KUKA KRL program: MyProgram_059().src

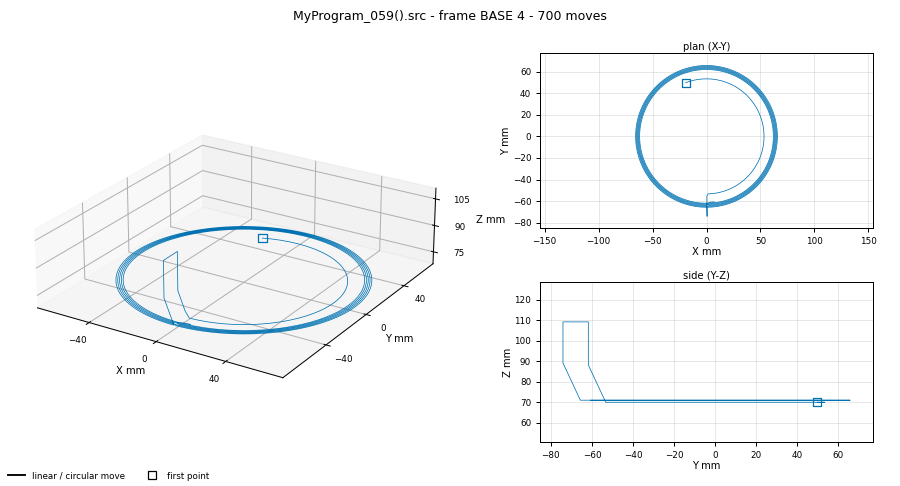
[picture p0: tool path of MyProgram_059().src in frame BASE 4, 700 of 700 moves have a stored position in this frame; points joined in program order, loops and branches not executed]
&ACCESS RVP
&REL 1
&PARAM TEMPLATE = C:\KRC\Roboter\Template\vorgabe
&PARAM EDITMASK = *
DEF MyProgram_059()
; ---- Setting reference (Base) ----
$BASE = BASE_DATA[4]

; --------------------------
; ---- Setting tool (TCP) ----
$TOOL = TOOL_DATA[3]
; --------------------------

$VEL.CP = VEL_APROX_PRINT
Startdeposition()
$VEL.CP = VEL_PRINT
LIN {X -19.2783,Y 49.7039,Z 70,A 103.8,B 24.8517,C -2.8098,E1 24.9442,E2 -20.1582} C_DIS
LIN {X -16.8217,Y 50.5882,Z 70,A 100.9889,B 24.8513,C -2.8131,E1 24.9516,E2 -17.3495} C_DIS
LIN {X -14.3168,Y 51.3533,Z 70,A 98.5431,B 24.8504,C -2.8223,E1 24.9581,E2 -14.9218} C_DIS
LIN {X -12.3251,Y 51.8679,Z 70,A 95.999,B 24.8507,C -2.8187,E1 24.9651,E2 -12.3655} C_DIS
LIN {X -9.9491,Y 52.3747,Z 70,A 93.3434,B 24.8506,C -2.8201,E1 24.9723,E2 -9.7102} C_DIS
LIN {X -7.1522,Y 52.8301,Z 70,A 90.3456,B 24.8503,C -2.8229,E1 24.9806,E2 -6.7165} C_DIS
LIN {X -4.5627,Y 53.1165,Z 70,A 87.5334,B 24.8502,C -2.8241,E1 24.9884,E2 -3.9056} C_DIS
LIN {X -2.028,Y 53.2732,Z 70,A 84.746,B 24.8502,C -2.8241,E1 24.9962,E2 -1.1173} C_DIS
LIN {X 0.6631,Y 53.308,Z 70,A 81.9222,B 24.85,C -2.8259,E1 25.0041,E2 1.7022} C_DIS
LIN {X 2.7693,Y 53.2395,Z 70,A 79.6668,B 24.85,C -2.8262,E1 25.0103,E2 3.9561} C_DIS
LIN {X 5.1925,Y 53.0585,Z 70,A 76.9708,B 24.8501,C -2.8244,E1 25.0178,E2 6.6547} C_DIS
LIN {X 7.8477,Y 52.7313,Z 70,A 74.1797,B 24.8501,C -2.8253,E1 25.0256,E2 9.4415} C_DIS
LIN {X 10.3045,Y 52.3063,Z 70,A 71.4304,B 24.8503,C -2.823,E1 25.0331,E2 12.1931} C_DIS
LIN {X 12.9755,Y 51.7089,Z 70,A 68.5235,B 24.8503,C -2.8221,E1 25.041,E2 15.0981} C_DIS
LIN {X 15.3915,Y 51.0415,Z 70,A 65.8321,B 24.8506,C -2.8203,E1 25.0482,E2 17.7892} C_DIS
LIN {X 17.8688,Y 50.2279,Z 70,A 63.0346,B 24.8508,C -2.818,E1 25.0556,E2 20.5865} C_DIS
LIN {X 20.3041,Y 49.2937,Z 70,A 60.2375,B 24.8511,C -2.8154,E1 25.0629,E2 23.3837} C_DIS
LIN {X 22.6903,Y 48.2418,Z 70,A 57.4092,B 24.8515,C -2.8117,E1 25.0701,E2 26.2135} C_DIS
LIN {X 25.039,Y 47.0657,Z 70,A 54.5794,B 24.8519,C -2.808,E1 25.0771,E2 29.0443} C_DIS
LIN {X 27.3333,Y 45.7715,Z 70,A 51.8043,B 24.8522,C -2.8051,E1 25.0838,E2 31.8179} C_DIS
LIN {X 29.6243,Y 44.3236,Z 70,A 48.9325,B 24.8526,C -2.8014,E1 25.0905,E2 34.6891} C_DIS
LIN {X 31.7582,Y 42.8206,Z 70,A 46.1065,B 24.8531,C -2.7963,E1 25.0969,E2 37.5173} C_DIS
LIN {X 33.7767,Y 41.2467,Z 70,A 43.3667,B 24.8536,C -2.7915,E1 25.1029,E2 40.2581} C_DIS
LIN {X 35.7658,Y 39.5343,Z 70,A 40.5427,B 24.8542,C -2.786,E1 25.1088,E2 43.0839} C_DIS
LIN {X 37.7091,Y 37.6855,Z 70,A 37.6907,B 24.8548,C -2.7807,E1 25.1145,E2 45.9366} C_DIS
LIN {X 39.4732,Y 35.8333,Z 70,A 34.9527,B 24.8554,C -2.775,E1 25.1197,E2 48.6762} C_DIS
LIN {X 41.1795,Y 33.8587,Z 70,A 32.1622,B 24.856,C -2.7689,E1 25.1248,E2 51.4684} C_DIS
LIN {X 42.8175,Y 31.7623,Z 70,A 29.318,B 24.8567,C -2.7624,E1 25.1296,E2 54.3145} C_DIS
LIN {X 44.3203,Y 29.6293,Z 70,A 26.559,B 24.8573,C -2.7563,E1 25.1339,E2 57.0741} C_DIS
LIN {X 45.6739,Y 27.496,Z 70,A 23.8275,B 24.8581,C -2.749,E1 25.138,E2 59.8092} C_DIS
LIN {X 46.9787,Y 25.202,Z 70,A 20.9748,B 24.8589,C -2.7411,E1 25.1418,E2 62.6655} C_DIS
LIN {X 48.1969,Y 22.7868,Z 70,A 18.1531,B 24.8595,C -2.7349,E1 25.1453,E2 65.4868} C_DIS
LIN {X 49.2137,Y 20.4974,Z 70,A 15.4462,B 24.8603,C -2.7271,E1 25.1483,E2 68.1975} C_DIS
LIN {X 50.191,Y 17.9733,Z 70,A 12.5854,B 24.8611,C -2.7197,E1 25.1511,E2 71.0598} C_DIS
LIN {X 50.9578,Y 15.6652,Z 70,A 10.2725,B 24.8612,C -2.7184,E1 25.153,E2 73.3627} C_DIS
LIN {X 51.5403,Y 13.6293,Z 70,A 7.7203,B 24.8625,C -2.7058,E1 25.1549,E2 75.9301} C_DIS
LIN {X 52.135,Y 11.1389,Z 70,A 4.9326,B 24.8634,C -2.6967,E1 25.1567,E2 78.7231} C_DIS
LIN {X 52.635,Y 8.4702,Z 70,A 2.0944,B 24.8642,C -2.6894,E1 25.158,E2 81.5619} C_DIS
LIN {X 52.9751,Y 5.9811,Z 70,A -0.6468,B 24.8651,C -2.6802,E1 25.159,E2 84.3088} C_DIS
LIN {X 53.2054,Y 3.3637,Z 70,A -3.419,B 24.8659,C -2.6724,E1 25.1596,E2 87.0828} C_DIS
LIN {X 53.3082,Y 0.6521,Z 70,A -6.2022,B 24.8665,C -2.6661,E1 25.1598,E2 89.8644} C_DIS
LIN {X 53.2792,Y -1.8589,Z 70,A -8.9946,B 24.8676,C -2.6556,E1 25.1596,E2 92.6651} C_DIS
LIN {X 53.1161,Y -4.5677,Z 70,A -11.8908,B 24.8685,C -2.6468,E1 25.159,E2 95.5648} C_DIS
LIN {X 52.84,Y -7.0759,Z 70,A -14.6152,B 24.8693,C -2.638,E1 25.1581,E2 98.294} C_DIS
LIN {X 52.4049,Y -9.7923,Z 70,A -17.5147,B 24.8701,C -2.6299,E1 25.1567,E2 101.1956} C_DIS
LIN {X 51.8877,Y -12.2395,Z 70,A -20.2234,B 24.871,C -2.6211,E1 25.1551,E2 103.9095} C_DIS
LIN {X 51.2007,Y -14.8551,Z 70,A -23.0427,B 24.8717,C -2.6139,E1 25.153,E2 106.7295} C_DIS
LIN {X 50.4138,Y -17.3388,Z 70,A -25.8264,B 24.8725,C -2.6057,E1 25.1505,E2 109.5169} C_DIS
LIN {X 49.5068,Y -19.7802,Z 70,A -28.6426,B 24.8734,C -2.5969,E1 25.1477,E2 112.3383} C_DIS
LIN {X 48.4704,Y -22.1994,Z 70,A -31.4173,B 24.8741,C -2.5896,E1 25.1446,E2 115.115} C_DIS
LIN {X 47.3664,Y -24.4654,Z 70,A -34.0954,B 24.8748,C -2.5824,E1 25.1412,E2 117.796} C_DIS
LIN {X 46.1668,Y -26.6593,Z 70,A -36.6069,B 24.8752,C -2.5784,E1 25.1378,E2 120.3037} C_DIS
LIN {X 45.0506,Y -28.5065,Z 70,A -39.1318,B 24.8762,C -2.5676,E1 25.1341,E2 122.8415} C_DIS
LIN {X 43.6375,Y -30.6252,Z 70,A -41.8671,B 24.877,C -2.5601,E1 25.1297,E2 125.5809} C_DIS
LIN {X 42.0253,Y -32.8034,Z 70,A -44.7117,B 24.8776,C -2.5538,E1 25.1249,E2 128.4269} C_DIS
LIN {X 40.4025,Y -34.7821,Z 70,A -47.4623,B 24.8782,C -2.5468,E1 25.12,E2 131.1815} C_DIS
LIN {X 38.6175,Y -36.7542,Z 70,A -50.3204,B 24.8789,C -2.5398,E1 25.1146,E2 134.0437} C_DIS
LIN {X 36.7529,Y -38.6187,Z 70,A -53.1054,B 24.8795,C -2.5341,E1 25.109,E2 136.8306} C_DIS
LIN {X 34.8576,Y -40.3374,Z 70,A -55.9121,B 24.8802,C -2.5267,E1 25.1031,E2 139.6435} C_DIS
LIN {X 32.6945,Y -42.1092,Z 70,A -58.8523,B 24.8806,C -2.5216,E1 25.0967,E2 142.5849} C_DIS
LIN {X 30.6521,Y -43.6188,Z 70,A -61.5165,B 24.881,C -2.5174,E1 25.0907,E2 145.2497} C_DIS
LIN {X 28.6394,Y -44.9655,Z 70,A -64.1754,B 24.8816,C -2.5112,E1 25.0844,E2 147.9144} C_DIS
LIN {X 26.3648,Y -46.3361,Z 70,A -67.0029,B 24.8821,C -2.5067,E1 25.0776,E2 150.744} C_DIS
LIN {X 23.9618,Y -47.6237,Z 70,A -69.8578,B 24.8824,C -2.5033,E1 25.0705,E2 153.599} C_DIS
LIN {X 21.667,Y -48.7102,Z 70,A -72.6403,B 24.8829,C -2.4981,E1 25.0635,E2 156.3868} C_DIS
LIN {X 19.2646,Y -49.7093,Z 70,A -75.4637,B 24.8833,C -2.4937,E1 25.0561,E2 159.2143} C_DIS
LIN {X 16.8142,Y -50.5907,Z 70,A -78.2509,B 24.8836,C -2.4904,E1 25.0488,E2 162.0037} C_DIS
LIN {X 14.3223,Y -51.3517,Z 70,A -81.0127,B 24.8838,C -2.4881,E1 25.0414,E2 164.7663} C_DIS
LIN {X 11.6989,Y -52.0126,Z 70,A -83.8932,B 24.884,C -2.4858,E1 25.0335,E2 167.6481} C_DIS
LIN {X 9.2126,Y -52.5096,Z 70,A -86.6359,B 24.8843,C -2.4833,E1 25.026,E2 170.3937} C_DIS
LIN {X 6.5156,Y -52.9125,Z 70,A -89.5294,B 24.8843,C -2.482,E1 25.018,E2 173.2876} C_DIS
LIN {X 4.0163,Y -53.1602,Z 70,A -92.2922,B 24.8846,C -2.4795,E1 25.0103,E2 176.0549} C_DIS
LIN {X 1.306,Y -53.2962,Z 70,A -95.144,B 24.8846,C -2.4797,E1 25.0024,E2 178.9055} C_DIS
LIN {X 1.306,Y -53.2962,Z 70,A -95.144,B 24.8846,C -2.4797,E1 25.0024,E2 178.9055} C_DIS
Enddeposition()
LIN {X 0.2997,Y -55.4223,Z 74.5315,A -95.1797,B 24.8832,C -2.4947,E1 25.0024,E2 178.9055} C_DIS
LIN {X 0.3807,Y -61.761,Z 88.1262,A -95.1515,B 24.8843,C -2.4828,E1 25.0024,E2 178.9055} C_DIS
LIN {X 0.3807,Y -61.761,Z 109.1262,A -95.5061,B 24.8699,C -2.632,E1 25.0024,E2 178.9055} C_DIS
LIN {X 0.5252,Y -74.1164,Z 109.1262,A -95.0495,B 24.8894,C -2.4276,E1 25.0023,E2 178.9347} C_DIS
LIN {X 0.5252,Y -74.1164,Z 89.1262,A -94.712,B 24.902,C -2.2856,E1 25.0023,E2 178.9347} C_DIS
LIN {X 0.4475,Y -67.7776,Z 75.5315,A -94.7382,B 24.901,C -2.2966,E1 25.0023,E2 178.9347} C_DIS
LIN {X 0.4215,Y -65.6646,Z 71,A -94.7484,B 24.9007,C -2.3009,E1 25.0023,E2 178.9347} C_DIS
Startdeposition()
$VEL.CP = VEL_PRINT
LIN {X -1.6116,Y -65.65,Z 71,A -97.5052,B 24.9027,C -2.2776,E1 24.9944,E2 181.7469} C_DIS
LIN {X -4.831,Y -65.4919,Z 71,A -100.3174,B 24.9027,C -2.2775,E1 24.9866,E2 184.5603} C_DIS
LIN {X -8.0387,Y -65.1759,Z 71,A -103.1307,B 24.9027,C -2.2778,E1 24.9788,E2 187.3746} C_DIS
LIN {X -11.227,Y -64.703,Z 71,A -105.9449,B 24.9027,C -2.2785,E1 24.971,E2 190.1896} C_DIS
LIN {X -14.3883,Y -64.0742,Z 71,A -108.76,B 24.9025,C -2.2797,E1 24.9633,E2 193.0054} C_DIS
LIN {X -17.515,Y -63.291,Z 71,A -111.5763,B 24.9024,C -2.2812,E1 24.9557,E2 195.8222} C_DIS
LIN {X -20.5994,Y -62.3553,Z 71,A -114.3935,B 24.9022,C -2.2832,E1 24.9482,E2 198.6397} C_DIS
LIN {X -23.6342,Y -61.2694,Z 71,A -117.2116,B 24.902,C -2.2855,E1 24.9408,E2 201.458} C_DIS
LIN {X -26.6121,Y -60.036,Z 71,A -120.0307,B 24.9018,C -2.2883,E1 24.9336,E2 204.277} C_DIS
LIN {X -29.5259,Y -58.6579,Z 71,A -122.8506,B 24.9015,C -2.2915,E1 24.9265,E2 207.0968} C_DIS
LIN {X -32.3685,Y -57.1384,Z 71,A -125.6715,B 24.9012,C -2.295,E1 24.9196,E2 209.9173} C_DIS
LIN {X -35.1332,Y -55.4814,Z 71,A -128.4933,B 24.9008,C -2.2989,E1 24.9129,E2 212.7386} C_DIS
LIN {X -37.8132,Y -53.6906,Z 71,A -131.316,B 24.9005,C -2.3032,E1 24.9064,E2 215.5606} C_DIS
LIN {X -40.4021,Y -51.7706,Z 71,A -134.1395,B 24.9001,C -2.3079,E1 24.9001,E2 218.3832} C_DIS
LIN {X -42.8937,Y -49.7258,Z 71,A -136.9639,B 24.8996,C -2.3129,E1 24.8941,E2 221.2066} C_DIS
LIN {X -45.282,Y -47.5612,Z 71,A -139.789,B 24.8992,C -2.3182,E1 24.8883,E2 224.0305} C_DIS
LIN {X -47.5612,Y -45.282,Z 71,A -142.615,B 24.8987,C -2.3238,E1 24.8828,E2 226.8551} C_DIS
LIN {X -49.7258,Y -42.8937,Z 71,A -145.4415,B 24.8982,C -2.3298,E1 24.8776,E2 229.6801} C_DIS
LIN {X -51.7706,Y -40.4021,Z 71,A -148.2689,B 24.8976,C -2.336,E1 24.8727,E2 232.5059} C_DIS
LIN {X -53.6906,Y -37.8132,Z 71,A -151.0969,B 24.897,C -2.3425,E1 24.868,E2 235.332} C_DIS
LIN {X -55.4814,Y -35.1332,Z 71,A -153.9254,B 24.8964,C -2.3493,E1 24.8637,E2 238.1586} C_DIS
LIN {X -57.1384,Y -32.3685,Z 71,A -156.7547,B 24.8958,C -2.3563,E1 24.8597,E2 240.9858} C_DIS
LIN {X -58.6579,Y -29.5259,Z 71,A -159.5844,B 24.8952,C -2.3636,E1 24.8561,E2 243.8133} C_DIS
LIN {X -60.036,Y -26.6121,Z 71,A -162.4148,B 24.8945,C -2.3711,E1 24.8528,E2 246.6413} C_DIS
LIN {X -61.2694,Y -23.6342,Z 71,A -165.2454,B 24.8938,C -2.3787,E1 24.8499,E2 249.4695} C_DIS
LIN {X -62.3553,Y -20.5994,Z 71,A -168.0766,B 24.8931,C -2.3866,E1 24.8473,E2 252.298} C_DIS
LIN {X -63.291,Y -17.515,Z 71,A -170.9079,B 24.8924,C -2.3945,E1 24.8451,E2 255.1266} C_DIS
LIN {X -64.0742,Y -14.3883,Z 71,A -173.7398,B 24.8917,C -2.4027,E1 24.8433,E2 257.9557} C_DIS
LIN {X -64.703,Y -11.227,Z 71,A -176.5719,B 24.8909,C -2.4109,E1 24.8418,E2 260.785} C_DIS
LIN {X -65.1759,Y -8.0387,Z 71,A -179.4041,B 24.8902,C -2.4192,E1 24.8408,E2 263.6141} C_DIS
LIN {X -65.4919,Y -4.831,Z 71,A 177.7633,B 24.8894,C -2.4276,E1 24.8401,E2 266.4436} C_DIS
LIN {X -65.65,Y -1.6116,Z 71,A 174.9641,B 24.8886,C -2.4367,E1 24.8398,E2 269.2379} C_DIS
LIN {X -65.65,Y 1.6116,Z 71,A 172.098,B 24.8878,C -2.4446,E1 24.8398,E2 272.1025} C_DIS
LIN {X -65.4919,Y 4.831,Z 71,A 169.2654,B 24.8871,C -2.4531,E1 24.8404,E2 274.9318} C_DIS
LIN {X -65.1759,Y 8.0387,Z 71,A 166.4326,B 24.8863,C -2.4616,E1 24.8412,E2 277.7613} C_DIS
LIN {X -64.703,Y 11.227,Z 71,A 163.6003,B 24.8855,C -2.4701,E1 24.8425,E2 280.5903} C_DIS
LIN {X -64.0742,Y 14.3883,Z 71,A 160.7677,B 24.8847,C -2.4785,E1 24.8441,E2 283.4194} C_DIS
LIN {X -63.291,Y 17.515,Z 71,A 157.9352,B 24.8839,C -2.4868,E1 24.8461,E2 286.2484} C_DIS
LIN {X -62.3553,Y 20.5994,Z 71,A 155.1031,B 24.8831,C -2.4951,E1 24.8485,E2 289.0771} C_DIS
LIN {X -61.2694,Y 23.6342,Z 71,A 152.2713,B 24.8824,C -2.5032,E1 24.8513,E2 291.9054} C_DIS
LIN {X -60.036,Y 26.6121,Z 71,A 149.4397,B 24.8816,C -2.5112,E1 24.8544,E2 294.7335} C_DIS
LIN {X -58.6579,Y 29.5259,Z 71,A 146.6086,B 24.8809,C -2.5191,E1 24.8578,E2 297.5612} C_DIS
LIN {X -57.1384,Y 32.3685,Z 71,A 143.7778,B 24.8801,C -2.5268,E1 24.8616,E2 300.3885} C_DIS
LIN {X -55.4814,Y 35.1332,Z 71,A 140.9475,B 24.8794,C -2.5343,E1 24.8658,E2 303.2153} C_DIS
LIN {X -53.6906,Y 37.8132,Z 71,A 138.1176,B 24.8787,C -2.5416,E1 24.8702,E2 306.0418} C_DIS
LIN {X -51.7706,Y 40.4021,Z 71,A 135.2883,B 24.8781,C -2.5486,E1 24.875,E2 308.8678} C_DIS
LIN {X -49.7258,Y 42.8937,Z 71,A 132.4596,B 24.8774,C -2.5555,E1 24.8801,E2 311.6932} C_DIS
LIN {X -47.5612,Y 45.282,Z 71,A 129.6314,B 24.8768,C -2.562,E1 24.8855,E2 314.5181} C_DIS
LIN {X -45.282,Y 47.5612,Z 71,A 126.8039,B 24.8762,C -2.5683,E1 24.8911,E2 317.3424} C_DIS
LIN {X -42.8937,Y 49.7258,Z 71,A 123.9773,B 24.8756,C -2.5743,E1 24.897,E2 320.1658} C_DIS
LIN {X -40.4021,Y 51.7706,Z 71,A 121.1511,B 24.875,C -2.58,E1 24.9032,E2 322.9889} C_DIS
LIN {X -37.8132,Y 53.6906,Z 71,A 118.3259,B 24.8745,C -2.5854,E1 24.9095,E2 325.8113} C_DIS
LIN {X -35.1332,Y 55.4814,Z 71,A 115.5014,B 24.874,C -2.5905,E1 24.9161,E2 328.6329} C_DIS
LIN {X -32.3685,Y 57.1384,Z 71,A 112.6776,B 24.8736,C -2.5952,E1 24.923,E2 331.4538} C_DIS
LIN {X -29.5259,Y 58.6579,Z 71,A 109.8548,B 24.8731,C -2.5996,E1 24.9299,E2 334.274} C_DIS
LIN {X -26.6121,Y 60.036,Z 71,A 107.0327,B 24.8727,C -2.6036,E1 24.9371,E2 337.0935} C_DIS
LIN {X -23.6342,Y 61.2694,Z 71,A 104.2116,B 24.8724,C -2.6072,E1 24.9444,E2 339.9122} C_DIS
LIN {X -20.5994,Y 62.3553,Z 71,A 101.3914,B 24.8721,C -2.6104,E1 24.9518,E2 342.7301} C_DIS
LIN {X -17.515,Y 63.291,Z 71,A 98.5723,B 24.8718,C -2.6133,E1 24.9594,E2 345.5471} C_DIS
LIN {X -14.3883,Y 64.0742,Z 71,A 95.7538,B 24.8715,C -2.6157,E1 24.967,E2 348.3635} C_DIS
LIN {X -11.227,Y 64.703,Z 71,A 92.9364,B 24.8713,C -2.6178,E1 24.9748,E2 351.179} C_DIS
LIN {X -8.0387,Y 65.1759,Z 71,A 90.1201,B 24.8712,C -2.6194,E1 24.9826,E2 353.9936} C_DIS
LIN {X -4.831,Y 65.4919,Z 71,A 87.3045,B 24.871,C -2.6207,E1 24.9904,E2 356.8075} C_DIS
LIN {X -1.6116,Y 65.65,Z 71,A 84.49,B 24.871,C -2.6215,E1 24.9982,E2 359.6206} C_DIS
LIN {X 1.6116,Y 65.65,Z 71,A 81.6766,B 24.871,C -2.6219,E1 25.0061,E2 362.4327} C_DIS
LIN {X 4.831,Y 65.4919,Z 71,A 78.8642,B 24.871,C -2.6219,E1 25.0139,E2 365.244} C_DIS
LIN {X 8.0387,Y 65.1759,Z 71,A 76.0526,B 24.871,C -2.6215,E1 25.0217,E2 368.0546} C_DIS
LIN {X 11.227,Y 64.703,Z 71,A 73.2421,B 24.871,C -2.6207,E1 25.0295,E2 370.8643} C_DIS
LIN {X 14.3883,Y 64.0742,Z 71,A 70.4326,B 24.8712,C -2.6194,E1 25.0371,E2 373.6731} C_DIS
LIN {X 17.515,Y 63.291,Z 71,A 67.6239,B 24.8713,C -2.6178,E1 25.0447,E2 376.4813} C_DIS
LIN {X 20.5994,Y 62.3553,Z 71,A 64.8162,B 24.8715,C -2.6157,E1 25.0522,E2 379.2887} C_DIS
LIN {X 23.6342,Y 61.2694,Z 71,A 62.0096,B 24.8718,C -2.6133,E1 25.0596,E2 382.0952} C_DIS
LIN {X 26.6121,Y 60.036,Z 71,A 59.2039,B 24.8721,C -2.6105,E1 25.0668,E2 384.9009} C_DIS
LIN {X 29.5259,Y 58.6579,Z 71,A 56.3998,B 24.8724,C -2.6073,E1 25.0738,E2 387.7053} C_DIS
LIN {X 32.3685,Y 57.1384,Z 71,A 53.5951,B 24.8727,C -2.6036,E1 25.0807,E2 390.5103} C_DIS
LIN {X 35.1332,Y 55.4814,Z 71,A 50.7919,B 24.8731,C -2.5997,E1 25.0873,E2 393.3141} C_DIS
LIN {X 37.8132,Y 53.6906,Z 71,A 47.9897,B 24.8735,C -2.5954,E1 25.0938,E2 396.1169} C_DIS
LIN {X 40.4021,Y 51.7706,Z 71,A 45.1883,B 24.874,C -2.5907,E1 25.1,E2 398.9192} C_DIS
LIN {X 42.8937,Y 49.7258,Z 71,A 42.3878,B 24.8745,C -2.5857,E1 25.106,E2 401.7208} C_DIS
LIN {X 45.282,Y 47.5612,Z 71,A 39.5878,B 24.875,C -2.5804,E1 25.1117,E2 404.522} C_DIS
LIN {X 47.5612,Y 45.282,Z 71,A 36.7888,B 24.8755,C -2.5747,E1 25.1172,E2 407.3223} C_DIS
LIN {X 49.7258,Y 42.8937,Z 71,A 33.9903,B 24.8761,C -2.5688,E1 25.1224,E2 410.1223} C_DIS
LIN {X 51.7706,Y 40.4021,Z 71,A 31.1928,B 24.8767,C -2.5626,E1 25.1273,E2 412.9215} C_DIS
LIN {X 53.6906,Y 37.8132,Z 71,A 28.3957,B 24.8773,C -2.5561,E1 25.1318,E2 415.7205} C_DIS
LIN {X 55.4814,Y 35.1332,Z 71,A 25.5992,B 24.878,C -2.5493,E1 25.1361,E2 418.5189} C_DIS
LIN {X 57.1384,Y 32.3685,Z 71,A 22.8032,B 24.8787,C -2.5424,E1 25.14,E2 421.317} C_DIS
LIN {X 58.6579,Y 29.5259,Z 71,A 20.0079,B 24.8794,C -2.5352,E1 25.1436,E2 424.1145} C_DIS
LIN {X 60.036,Y 26.6121,Z 71,A 17.213,B 24.8801,C -2.5278,E1 25.1469,E2 426.9118} C_DIS
LIN {X 61.2694,Y 23.6342,Z 71,A 14.4184,B 24.8808,C -2.5202,E1 25.1498,E2 429.7088} C_DIS
LIN {X 62.3553,Y 20.5994,Z 71,A 11.6243,B 24.8815,C -2.5124,E1 25.1523,E2 432.5055} C_DIS
LIN {X 63.291,Y 17.515,Z 71,A 8.8307,B 24.8823,C -2.5045,E1 25.1545,E2 435.3018} C_DIS
LIN {X 64.0742,Y 14.3883,Z 71,A 6.0374,B 24.883,C -2.4965,E1 25.1563,E2 438.0979} C_DIS
LIN {X 64.703,Y 11.227,Z 71,A 3.244,B 24.8838,C -2.4884,E1 25.1578,E2 440.8942} C_DIS
LIN {X 65.1759,Y 8.0387,Z 71,A 0.4512,B 24.8845,C -2.4801,E1 25.1588,E2 443.69} C_DIS
LIN {X 65.4919,Y 4.831,Z 71,A -2.3417,B 24.8853,C -2.4718,E1 25.1595,E2 446.4859} C_DIS
LIN {X 65.65,Y 1.6116,Z 71,A -5.0201,B 24.8858,C -2.4664,E1 25.1598,E2 449.1611} C_DIS
LIN {X 65.65,Y -1.6116,Z 71,A -7.9269,B 24.8869,C -2.4551,E1 25.1597,E2 452.0775} C_DIS
LIN {X 65.4919,Y -4.831,Z 71,A -10.7193,B 24.8877,C -2.4467,E1 25.1592,E2 454.8732} C_DIS
LIN {X 65.1759,Y -8.0387,Z 71,A -13.512,B 24.8884,C -2.4383,E1 25.1583,E2 457.6691} C_DIS
LIN {X 64.703,Y -11.227,Z 71,A -16.3045,B 24.8892,C -2.4299,E1 25.1571,E2 460.4651} C_DIS
LIN {X 64.0742,Y -14.3883,Z 71,A -19.0971,B 24.8899,C -2.4216,E1 25.1555,E2 463.2611} C_DIS
LIN {X 63.291,Y -17.515,Z 71,A -21.8901,B 24.8907,C -2.4133,E1 25.1535,E2 466.0575} C_DIS
LIN {X 62.3553,Y -20.5994,Z 71,A -24.6832,B 24.8914,C -2.4052,E1 25.1511,E2 468.8541} C_DIS
LIN {X 61.2694,Y -23.6342,Z 71,A -27.4766,B 24.8922,C -2.3971,E1 25.1484,E2 471.6509} C_DIS
LIN {X 60.036,Y -26.6121,Z 71,A -30.2702,B 24.8929,C -2.3891,E1 25.1454,E2 474.4479} C_DIS
LIN {X 58.6579,Y -29.5259,Z 71,A -33.0641,B 24.8936,C -2.3813,E1 25.1419,E2 477.2453} C_DIS
LIN {X 57.1384,Y -32.3685,Z 71,A -35.8584,B 24.8943,C -2.3737,E1 25.1382,E2 480.0431} C_DIS
LIN {X 55.4814,Y -35.1332,Z 71,A -38.6532,B 24.8949,C -2.3663,E1 25.1341,E2 482.8413} C_DIS
LIN {X 53.6906,Y -37.8132,Z 71,A -41.4485,B 24.8956,C -2.359,E1 25.1296,E2 485.64} C_DIS
LIN {X 51.7706,Y -40.4021,Z 71,A -44.2442,B 24.8962,C -2.3519,E1 25.1249,E2 488.4391} C_DIS
LIN {X 49.7258,Y -42.8937,Z 71,A -47.0406,B 24.8968,C -2.3451,E1 25.1199,E2 491.2388} C_DIS
LIN {X 47.5612,Y -45.282,Z 71,A -49.8374,B 24.8974,C -2.3386,E1 25.1146,E2 494.0389} C_DIS
LIN {X 45.282,Y -47.5612,Z 71,A -52.635,B 24.8979,C -2.3323,E1 25.109,E2 496.8397} C_DIS
LIN {X 42.8937,Y -49.7258,Z 71,A -55.4332,B 24.8985,C -2.3263,E1 25.1031,E2 499.6409} C_DIS
LIN {X 40.4021,Y -51.7706,Z 71,A -58.2322,B 24.899,C -2.3205,E1 25.097,E2 502.4429} C_DIS
LIN {X 37.8132,Y -53.6906,Z 71,A -61.0317,B 24.8994,C -2.3151,E1 25.0907,E2 505.2455} C_DIS
LIN {X 35.1332,Y -55.4814,Z 71,A -63.8321,B 24.8999,C -2.31,E1 25.0841,E2 508.0487} C_DIS
LIN {X 32.3685,Y -57.1384,Z 71,A -66.6334,B 24.9003,C -2.3052,E1 25.0773,E2 510.8528} C_DIS
LIN {X 29.5259,Y -58.6579,Z 71,A -69.4353,B 24.9007,C -2.3008,E1 25.0704,E2 513.6574} C_DIS
LIN {X 26.6121,Y -60.036,Z 71,A -72.2383,B 24.901,C -2.2968,E1 25.0633,E2 516.4629} C_DIS
LIN {X 23.6342,Y -61.2694,Z 71,A -75.042,B 24.9013,C -2.2931,E1 25.056,E2 519.269} C_DIS
LIN {X 20.5994,Y -62.3553,Z 71,A -77.8466,B 24.9016,C -2.2897,E1 25.0486,E2 522.076} C_DIS
LIN {X 17.515,Y -63.291,Z 71,A -80.652,B 24.9019,C -2.2868,E1 25.0411,E2 524.8836} C_DIS
LIN {X 14.3883,Y -64.0742,Z 71,A -83.4585,B 24.9021,C -2.2843,E1 25.0334,E2 527.6922} C_DIS
LIN {X 11.227,Y -64.703,Z 71,A -86.266,B 24.9023,C -2.2821,E1 25.0257,E2 530.5016} C_DIS
LIN {X 8.0387,Y -65.1759,Z 71,A -89.0742,B 24.9024,C -2.2804,E1 25.0179,E2 533.3115} C_DIS
LIN {X 4.831,Y -65.4919,Z 71,A -91.8836,B 24.9026,C -2.279,E1 25.0101,E2 536.1226} C_DIS
LIN {X 1.6116,Y -65.65,Z 71,A -94.6939,B 24.9026,C -2.2781,E1 25.0023,E2 538.9343} C_DIS
LIN {X 1.6116,Y -65.65,Z 71,A -94.6939,B 24.9026,C -2.2781,E1 25.0023,E2 538.9343} C_DIS
Enddeposition()
LIN {X 0.4182,Y -64.7452,Z 71,A -95.2534,B 24.9003,C -2.3051,E1 25.0009,E2 539.4297} C_DIS
Startdeposition()
$VEL.CP = VEL_PRINT
LIN {X 1.7046,Y -64.7278,Z 71,A -93.2371,B 24.8985,C -2.3258,E1 25.0067,E2 537.3646} C_DIS
LIN {X 4.8039,Y -64.5722,Z 71,A -90.5664,B 24.8985,C -2.3252,E1 25.0141,E2 534.6964} C_DIS
LIN {X 7.9677,Y -64.2586,Z 71,A -87.7742,B 24.8985,C -2.3263,E1 25.0218,E2 531.9035} C_DIS
LIN {X 10.9714,Y -63.8141,Z 71,A -84.9741,B 24.8981,C -2.331,E1 25.0296,E2 529.0951} C_DIS
LIN {X 14.2629,Y -63.1601,Z 71,A -81.7635,B 24.8973,C -2.3394,E1 25.0384,E2 525.8687} C_DIS
LIN {X 18.0954,Y -62.1706,Z 71,A -78.6805,B 24.8979,C -2.333,E1 25.0466,E2 522.806} C_DIS
LIN {X 20.7104,Y -61.3482,Z 71,A -76.286,B 24.8977,C -2.3351,E1 25.053,E2 520.4108} C_DIS
LIN {X 23.4358,Y -60.3602,Z 71,A -73.7752,B 24.8975,C -2.3372,E1 25.0596,E2 517.9005} C_DIS
LIN {X 25.9705,Y -59.3133,Z 71,A -71.2966,B 24.8971,C -2.342,E1 25.0659,E2 515.4165} C_DIS
LIN {X 28.3807,Y -58.1996,Z 71,A -68.8888,B 24.8966,C -2.3471,E1 25.072,E2 513.0027} C_DIS
LIN {X 30.6809,Y -57.019,Z 71,A -66.5457,B 24.8962,C -2.3523,E1 25.0778,E2 510.6538} C_DIS
LIN {X 33.4449,Y -55.4437,Z 71,A -63.7576,B 24.8958,C -2.3567,E1 25.0845,E2 507.8639} C_DIS
LIN {X 36.4079,Y -53.5443,Z 71,A -60.9837,B 24.896,C -2.3542,E1 25.091,E2 505.1051} C_DIS
LIN {X 38.9266,Y -51.7421,Z 71,A -57.6008,B 24.8941,C -2.376,E1 25.0987,E2 501.6826} C_DIS
LIN {X 42.5093,Y -48.8415,Z 71,A -53.924,B 24.8941,C -2.3748,E1 25.1065,E2 498.0229} C_DIS
LIN {X 44.7414,Y -46.806,Z 71,A -51.6708,B 24.8946,C -2.3703,E1 25.1111,E2 495.7894} C_DIS
LIN {X 46.6065,Y -44.9483,Z 71,A -48.6884,B 24.8926,C -2.3926,E1 25.117,E2 492.767} C_DIS
LIN {X 49.1133,Y -42.1949,Z 71,A -44.7946,B 24.8904,C -2.4164,E1 25.1242,E2 488.8344} C_DIS
LIN {X 51.3927,Y -39.3871,Z 71,A -42.8171,B 24.8925,C -2.3932,E1 25.1275,E2 486.9212} C_DIS
LIN {X 53.2141,Y -36.8889,Z 71,A -39.7779,B 24.8911,C -2.4084,E1 25.1325,E2 483.8607} C_DIS
LIN {X 54.7989,Y -34.4913,Z 71,A -37.3202,B 24.8907,C -2.4132,E1 25.1362,E2 481.4039} C_DIS
LIN {X 56.3728,Y -31.8549,Z 71,A -34.6384,B 24.8901,C -2.4201,E1 25.14,E2 478.7198} C_DIS
LIN {X 57.8193,Y -29.1476,Z 71,A -31.8327,B 24.8892,C -2.4303,E1 25.1436,E2 475.9048} C_DIS
LIN {X 59.1158,Y -26.4175,Z 71,A -29.2185,B 24.8886,C -2.4367,E1 25.1467,E2 473.2897} C_DIS
LIN {X 60.2296,Y -23.7681,Z 71,A -26.7325,B 24.888,C -2.4428,E1 25.1493,E2 470.8028} C_DIS
LIN {X 61.2059,Y -21.1297,Z 71,A -24.1636,B 24.8871,C -2.4525,E1 25.1517,E2 468.2255} C_DIS
LIN {X 62.2491,Y -17.8213,Z 71,A -21.2378,B 24.8866,C -2.4582,E1 25.1541,E2 465.3028} C_DIS
LIN {X 63.0327,Y -14.8142,Z 71,A -18.4724,B 24.8857,C -2.4672,E1 25.1559,E2 462.5321} C_DIS
LIN {X 63.6504,Y -11.8858,Z 71,A -15.7461,B 24.8848,C -2.4776,E1 25.1574,E2 459.7972} C_DIS
LIN {X 64.1177,Y -9.0246,Z 71,A -13.2664,B 24.8842,C -2.4835,E1 25.1585,E2 457.3183} C_DIS
LIN {X 64.4061,Y -6.6623,Z 71,A -11.1444,B 24.8836,C -2.4906,E1 25.1591,E2 455.1921} C_DIS
LIN {X 64.6484,Y -3.6211,Z 71,A -8.6199,B 24.8832,C -2.4945,E1 25.1596,E2 452.6732} C_DIS
LIN {X 64.7426,Y -0.9786,Z 71,A -6.2071,B 24.8823,C -2.5038,E1 25.1598,E2 450.2528} C_DIS
LIN {X 64.724,Y 1.8298,Z 71,A -3.7054,B 24.8815,C -2.5121,E1 25.1597,E2 447.7463} C_DIS
LIN {X 64.5772,Y 4.7381,Z 71,A -1.1277,B 24.8808,C -2.5202,E1 25.1592,E2 445.1648} C_DIS
LIN {X 64.2984,Y 7.6322,Z 71,A 1.3576,B 24.8802,C -2.526,E1 25.1585,E2 442.6806} C_DIS
LIN {X 63.92,Y 10.3377,Z 71,A 3.8525,B 24.8793,C -2.5355,E1 25.1574,E2 440.1779} C_DIS
LIN {X 63.4025,Y 13.1401,Z 71,A 6.1121,B 24.8793,C -2.5364,E1 25.1562,E2 437.9293} C_DIS
LIN {X 62.7673,Y 15.901,Z 71,A 8.8141,B 24.878,C -2.5491,E1 25.1544,E2 435.2131} C_DIS
LIN {X 61.9824,Y 18.7299,Z 71,A 11.4389,B 24.8772,C -2.5575,E1 25.1524,E2 432.5833} C_DIS
LIN {X 61.1425,Y 21.3105,Z 71,A 13.8102,B 24.8766,C -2.5638,E1 25.1503,E2 430.2106} C_DIS
LIN {X 59.5888,Y 25.3321,Z 71,A 18.3697,B 24.8737,C -2.594,E1 25.1454,E2 425.6049} C_DIS
LIN {X 58.1806,Y 28.4198,Z 71,A 20.9945,B 24.8738,C -2.5924,E1 25.1422,E2 422.9978} C_DIS
LIN {X 56.3655,Y 31.868,Z 71,A 23.9965,B 24.874,C -2.5901,E1 25.1382,E2 420.0168} C_DIS
LIN {X 54.9804,Y 34.2007,Z 71,A 26.2226,B 24.8739,C -2.5919,E1 25.135,E2 417.7978} C_DIS
LIN {X 53.6459,Y 36.258,Z 71,A 28.5043,B 24.8731,C -2.6003,E1 25.1315,E2 415.5078} C_DIS
LIN {X 51.9591,Y 38.6377,Z 71,A 31.0957,B 24.8724,C -2.6068,E1 25.1272,E2 412.9135} C_DIS
LIN {X 50.0806,Y 41.0436,Z 71,A 33.5523,B 24.8724,C -2.607,E1 25.123,E2 410.468} C_DIS
LIN {X 48.6103,Y 42.774,Z 71,A 35.729,B 24.8715,C -2.6157,E1 25.119,E2 408.2804} C_DIS
LIN {X 46.7235,Y 44.8269,Z 71,A 38.148,B 24.8711,C -2.6199,E1 25.1144,E2 405.8621} C_DIS
LIN {X 44.7407,Y 46.8067,Z 71,A 40.7361,B 24.8704,C -2.6277,E1 25.1092,E2 403.2663} C_DIS
LIN {X 42.662,Y 48.7081,Z 71,A 43.0721,B 24.8703,C -2.6287,E1 25.1043,E2 400.9374} C_DIS
LIN {X 40.8961,Y 50.2002,Z 71,A 45.2368,B 24.8696,C -2.6354,E1 25.0997,E2 398.765} C_DIS
LIN {X 38.2913,Y 52.214,Z 71,A 48.0947,B 24.8692,C -2.6391,E1 25.0933,E2 395.9086} C_DIS
LIN {X 36.0765,Y 53.7688,Z 71,A 50.6553,B 24.8684,C -2.6471,E1 25.0874,E2 393.3379} C_DIS
LIN {X 33.3903,Y 55.4769,Z 71,A 53.6606,B 24.8676,C -2.6558,E1 25.0802,E2 390.3213} C_DIS
LIN {X 29.2381,Y 57.773,Z 71,A 57.5697,B 24.8677,C -2.6543,E1 25.0706,E2 386.4268} C_DIS
LIN {X 26.6486,Y 59.0117,Z 71,A 60.6859,B 24.866,C -2.6711,E1 25.0626,E2 383.2787} C_DIS
LIN {X 22.6001,Y 60.6785,Z 71,A 63.9633,B 24.8671,C -2.6605,E1 25.0542,E2 380.0336} C_DIS
LIN {X 19.5784,Y 61.7199,Z 71,A 66.7843,B 24.8669,C -2.6627,E1 25.0467,E2 377.213} C_DIS
LIN {X 16.944,Y 62.4934,Z 71,A 69.4569,B 24.8661,C -2.67,E1 25.0395,E2 374.5273} C_DIS
LIN {X 13.3255,Y 63.3644,Z 71,A 72.463,B 24.8666,C -2.6649,E1 25.0313,E2 371.5374} C_DIS
LIN {X 10.1955,Y 63.9427,Z 71,A 75.2599,B 24.8666,C -2.6654,E1 25.0236,E2 368.7421} C_DIS
LIN {X 7.1086,Y 64.3593,Z 71,A 78.1134,B 24.8663,C -2.6682,E1 25.0157,E2 365.8843} C_DIS
LIN {X 4.3371,Y 64.6043,Z 71,A 80.5068,B 24.8665,C -2.6668,E1 25.0091,E2 363.4955} C_DIS
LIN {X 1.3797,Y 64.7352,Z 71,A 83.1186,B 24.8665,C -2.6663,E1 25.0018,E2 360.8853} C_DIS
LIN {X -1.4518,Y 64.7339,Z 71,A 85.573,B 24.8667,C -2.6646,E1 24.9949,E2 358.435} C_DIS
LIN {X -3.7949,Y 64.6387,Z 71,A 87.4954,B 24.8671,C -2.6605,E1 24.9896,E2 356.5219} C_DIS
LIN {X -6.7317,Y 64.3988,Z 71,A 90.3265,B 24.8667,C -2.6642,E1 24.9817,E2 353.6805} C_DIS
LIN {X -9.7832,Y 64.0064,Z 71,A 93.0266,B 24.8669,C -2.662,E1 24.9742,E2 350.9836} C_DIS
LIN {X -12.7851,Y 63.4753,Z 71,A 95.3182,B 24.868,C -2.651,E1 24.968,E2 348.7155} C_DIS
LIN {X -15.7442,Y 62.8075,Z 71,A 98.4837,B 24.8672,C -2.659,E1 24.9593,E2 345.5269} C_DIS
LIN {X -17.7054,Y 62.2819,Z 71,A 100.8122,B 24.8663,C -2.6687,E1 24.953,E2 343.1716} C_DIS
LIN {X -23.039,Y 60.5123,Z 71,A 105.1796,B 24.8682,C -2.6495,E1 24.9416,E2 338.8414} C_DIS
LIN {X -26.227,Y 59.2012,Z 71,A 108.3051,B 24.8685,C -2.6468,E1 24.9336,E2 335.7151} C_DIS
LIN {X -29.0462,Y 57.87,Z 71,A 111.1049,B 24.8688,C -2.6433,E1 24.9266,E2 332.9162} C_DIS
LIN {X -31.9315,Y 56.3298,Z 71,A 113.9617,B 24.8694,C -2.6376,E1 24.9196,E2 330.0648} C_DIS
LIN {X -34.253,Y 54.9477,Z 71,A 116.3641,B 24.8698,C -2.6336,E1 24.9139,E2 327.6646} C_DIS
LIN {X -36.7619,Y 53.3024,Z 71,A 118.9989,B 24.8703,C -2.628,E1 24.9078,E2 325.0343} C_DIS
LIN {X -39.0605,Y 51.6415,Z 71,A 121.5005,B 24.8708,C -2.6228,E1 24.9022,E2 322.5364} C_DIS
LIN {X -41.1794,Y 49.9684,Z 71,A 123.8801,B 24.8714,C -2.6175,E1 24.897,E2 320.1605} C_DIS
LIN {X -43.4347,Y 48.0214,Z 71,A 126.6046,B 24.8718,C -2.6134,E1 24.8913,E2 317.435} C_DIS
LIN {X -45.3138,Y 46.252,Z 71,A 128.8983,B 24.8723,C -2.6082,E1 24.8867,E2 315.144} C_DIS
LIN {X -47.3288,Y 44.1878,Z 71,A 131.4144,B 24.873,C -2.6013,E1 24.8818,E2 312.6335} C_DIS
LIN {X -49.1204,Y 42.1874,Z 71,A 133.7786,B 24.8736,C -2.5951,E1 24.8775,E2 310.2734} C_DIS
LIN {X -50.821,Y 40.1216,Z 71,A 136.2745,B 24.8739,C -2.5916,E1 24.8731,E2 307.7743} C_DIS
LIN {X -52.7947,Y 37.4868,Z 71,A 139.1809,B 24.8747,C -2.5837,E1 24.8684,E2 304.8727} C_DIS
LIN {X -54.4809,Y 34.9908,Z 71,A 141.8639,B 24.8754,C -2.5767,E1 24.8642,E2 302.1929} C_DIS
LIN {X -56.0788,Y 32.3682,Z 71,A 144.1363,B 24.8769,C -2.5603,E1 24.861,E2 299.9481} C_DIS
LIN {X -57.937,Y 28.9099,Z 71,A 147.822,B 24.8775,C -2.5544,E1 24.8562,E2 296.2569} C_DIS
LIN {X -59.3194,Y 25.9565,Z 71,A 151.0152,B 24.8777,C -2.5519,E1 24.8525,E2 293.0522} C_DIS
LIN {X -60.2724,Y 23.6591,Z 71,A 154.3976,B 24.8761,C -2.5688,E1 24.849,E2 289.6105} C_DIS
LIN {X -61.7309,Y 19.5439,Z 71,A 157.0665,B 24.8795,C -2.5332,E1 24.8467,E2 287.0114} C_DIS
LIN {X -62.9701,Y 15.0786,Z 71,A 161.2263,B 24.8806,C -2.5216,E1 24.8438,E2 282.855} C_DIS
LIN {X -63.5958,Y 12.1694,Z 71,A 163.6078,B 24.8819,C -2.5085,E1 24.8424,E2 280.4909} C_DIS
LIN {X -64.0698,Y 9.3617,Z 71,A 166.4267,B 24.8821,C -2.5063,E1 24.8412,E2 277.6603} C_DIS
LIN {X -64.444,Y 6.2933,Z 71,A 169.1697,B 24.8829,C -2.4978,E1 24.8404,E2 274.9212} C_DIS
LIN {X -64.6718,Y 3.1974,Z 71,A 171.9795,B 24.8836,C -2.4904,E1 24.8399,E2 272.1124} C_DIS
LIN {X -64.7516,Y 0.0903,Z 71,A 174.592,B 24.8847,C -2.479,E1 24.8398,E2 269.5113} C_DIS
LIN {X -64.7034,Y -2.4675,Z 71,A 176.9247,B 24.8852,C -2.4732,E1 24.84,E2 267.1784} C_DIS
LIN {X -64.5414,Y -5.1888,Z 71,A 179.402,B 24.8858,C -2.4669,E1 24.8405,E2 264.7011} C_DIS
LIN {X -64.2485,Y -8.0456,Z 71,A -177.9905,B 24.8864,C -2.4603,E1 24.8413,E2 262.0939} C_DIS
LIN {X -63.7656,Y -11.248,Z 71,A -175.2201,B 24.8874,C -2.4496,E1 24.8425,E2 259.3326} C_DIS
LIN {X -62.9577,Y -15.1294,Z 71,A -170.9813,B 24.887,C -2.4535,E1 24.8452,E2 255.0596} C_DIS
LIN {X -60.7937,Y -22.2859,Z 71,A -165.0221,B 24.89,C -2.4208,E1 24.8502,E2 249.1443} C_DIS
LIN {X -59.7902,Y -24.8547,Z 71,A -162.6078,B 24.8907,C -2.4133,E1 24.8527,E2 246.7344} C_DIS
LIN {X -58.8049,Y -27.1029,Z 71,A -160.377,B 24.8911,C -2.4085,E1 24.8553,E2 244.5031} C_DIS
LIN {X -57.4565,Y -29.8562,Z 71,A -157.5218,B 24.8916,C -2.4039,E1 24.8589,E2 241.6433} C_DIS
LIN {X -55.9716,Y -32.5548,Z 71,A -154.3232,B 24.8913,C -2.4064,E1 24.8633,E2 238.4222} C_DIS
LIN {X -53.8094,Y -36.0164,Z 71,A -151.133,B 24.8929,C -2.3886,E1 24.8681,E2 235.2583} C_DIS
LIN {X -52.0541,Y -38.5097,Z 71,A -148.5165,B 24.8937,C -2.3804,E1 24.8724,E2 232.6487} C_DIS
LIN {X -50.057,Y -41.0724,Z 71,A -145.6049,B 24.8942,C -2.3744,E1 24.8775,E2 229.7377} C_DIS
LIN {X -48.3145,Y -43.1073,Z 71,A -143.2226,B 24.8947,C -2.3694,E1 24.8819,E2 227.3567} C_DIS
LIN {X -46.2862,Y -45.2792,Z 71,A -140.6531,B 24.8953,C -2.3625,E1 24.8868,E2 224.7924} C_DIS
LIN {X -44.0848,Y -47.4255,Z 71,A -137.8416,B 24.8956,C -2.3589,E1 24.8925,E2 221.9779} C_DIS
LIN {X -41.7817,Y -49.466,Z 71,A -134.8115,B 24.8955,C -2.3603,E1 24.8989,E2 218.9328} C_DIS
LIN {X -39.0069,Y -51.6817,Z 71,A -132.2407,B 24.897,C -2.3426,E1 24.9045,E2 216.3946} C_DIS
LIN {X -37.2721,Y -52.9476,Z 71,A -129.958,B 24.8966,C -2.3476,E1 24.9098,E2 214.0922} C_DIS
LIN {X -34.6917,Y -54.6728,Z 71,A -127.2262,B 24.897,C -2.343,E1 24.9162,E2 211.3623} C_DIS
LIN {X -32.1145,Y -56.2246,Z 71,A -124.6148,B 24.8974,C -2.3382,E1 24.9224,E2 208.7545} C_DIS
LIN {X -29.261,Y -57.7613,Z 71,A -121.1086,B 24.8965,C -2.3486,E1 24.9312,E2 205.214} C_DIS
LIN {X -25.3652,Y -59.575,Z 71,A -117.9088,B 24.898,C -2.3312,E1 24.9393,E2 202.048} C_DIS
LIN {X -22.6064,Y -60.6761,Z 71,A -115.2392,B 24.8982,C -2.3297,E1 24.9463,E2 199.3764} C_DIS
LIN {X -19.7341,Y -61.6695,Z 71,A -112.3189,B 24.8979,C -2.3328,E1 24.954,E2 196.4433} C_DIS
LIN {X -16.4519,Y -62.6257,Z 71,A -109.4408,B 24.8983,C -2.3276,E1 24.9618,E2 193.5732} C_DIS
LIN {X -13.2989,Y -63.3699,Z 71,A -106.7714,B 24.8989,C -2.3218,E1 24.969,E2 190.9142} C_DIS
LIN {X -10.6775,Y -63.8632,Z 71,A -104.3414,B 24.8988,C -2.3226,E1 24.9757,E2 188.4797} C_DIS
LIN {X -7.9404,Y -64.262,Z 71,A -101.7675,B 24.8986,C -2.325,E1 24.9829,E2 185.8982} C_DIS
LIN {X -4.8281,Y -64.5703,Z 71,A -99.0509,B 24.8986,C -2.3237,E1 24.9904,E2 183.1834} C_DIS
LIN {X -1.6904,Y -64.7283,Z 71,A -96.4043,B 24.8989,C -2.3209,E1 24.9978,E2 180.5429} C_DIS
LIN {X 0.4182,Y -64.7452,Z 71,A -95.2529,B 24.9003,C -2.3049,E1 25.0009,E2 179.4297} C_DIS
Enddeposition()
LIN {X 0.4182,Y -64.7452,Z 71,A -95.2529,B 24.9003,C -2.3049,E1 25.0009,E2 179.4297} C_DIS
Startdeposition()
$VEL.CP = VEL_PRINT
LIN {X -1.1857,Y -63.8198,Z 71,A -97.1822,B 24.8999,C -2.3095,E1 24.9955,E2 181.348} C_DIS
LIN {X -4.0145,Y -63.7051,Z 71,A -99.6752,B 24.8999,C -2.3104,E1 24.9886,E2 183.8395} C_DIS
LIN {X -8.3643,Y -63.2806,Z 71,A -103.697,B 24.8999,C -2.3087,E1 24.9774,E2 187.8679} C_DIS
LIN {X -11.277,Y -62.8267,Z 71,A -106.2717,B 24.8998,C -2.311,E1 24.9703,E2 190.4394} C_DIS
LIN {X -14.1334,Y -62.2469,Z 71,A -109.0904,B 24.9001,C -2.3078,E1 24.9626,E2 193.2693} C_DIS
LIN {X -17.292,Y -61.444,Z 71,A -112.8662,B 24.9015,C -2.2915,E1 24.9523,E2 197.0897} C_DIS
LIN {X -20.9523,Y -60.2943,Z 71,A -115.3062,B 24.8994,C -2.3155,E1 24.946,E2 199.4773} C_DIS
LIN {X -24.2181,Y -59.0578,Z 71,A -118.3543,B 24.899,C -2.3203,E1 24.9381,E2 202.5206} C_DIS
LIN {X -26.7747,Y -57.9432,Z 71,A -121.16,B 24.8993,C -2.3167,E1 24.9309,E2 205.3417} C_DIS
LIN {X -29.8731,Y -56.4091,Z 71,A -124.0518,B 24.8986,C -2.3249,E1 24.9237,E2 208.2217} C_DIS
LIN {X -31.6034,Y -55.4585,Z 71,A -125.8142,B 24.8984,C -2.3275,E1 24.9195,E2 209.983} C_DIS
LIN {X -33.9838,Y -54.0325,Z 71,A -128.3353,B 24.8981,C -2.3305,E1 24.9135,E2 212.5048} C_DIS
LIN {X -36.3492,Y -52.4701,Z 71,A -131.2681,B 24.8984,C -2.3266,E1 24.9066,E2 215.4567} C_DIS
LIN {X -41.0022,Y -48.921,Z 71,A -135.95,B 24.8966,C -2.3475,E1 24.8964,E2 220.106} C_DIS
LIN {X -42.6722,Y -47.4708,Z 71,A -138.1831,B 24.8966,C -2.3464,E1 24.8917,E2 222.3507} C_DIS
LIN {X -45.8173,Y -44.443,Z 71,A -141.8668,B 24.8956,C -2.3591,E1 24.8844,E2 226.0195} C_DIS
LIN {X -47.435,Y -42.7121,Z 71,A -144.6439,B 24.8963,C -2.3509,E1 24.8791,E2 228.8286} C_DIS
LIN {X -50.2116,Y -39.4107,Z 71,A -148.2031,B 24.895,C -2.3659,E1 24.8729,E2 232.3683} C_DIS
LIN {X -52.076,Y -36.912,Z 71,A -151.1465,B 24.8946,C -2.3699,E1 24.8681,E2 235.3165} C_DIS
LIN {X -53.5417,Y -34.7528,Z 71,A -154.0447,B 24.895,C -2.3651,E1 24.8636,E2 238.2409} C_DIS
LIN {X -56.0047,Y -30.6249,Z 71,A -157.6486,B 24.8928,C -2.3901,E1 24.8587,E2 241.8038} C_DIS
LIN {X -57.4204,Y -27.8807,Z 71,A -160.6529,B 24.8925,C -2.3932,E1 24.8549,E2 244.8169} C_DIS
LIN {X -58.6589,Y -25.1721,Z 71,A -162.8314,B 24.891,C -2.4102,E1 24.8525,E2 246.9668} C_DIS
LIN {X -59.3747,Y -23.4313,Z 71,A -164.8483,B 24.8911,C -2.4087,E1 24.8503,E2 248.9984} C_DIS
LIN {X -61.1502,Y -18.3044,Z 71,A -169.5656,B 24.8896,C -2.4259,E1 24.8462,E2 253.7016} C_DIS
LIN {X -61.8914,Y -15.6157,Z 71,A -172.2896,B 24.8893,C -2.4292,E1 24.8442,E2 256.4336} C_DIS
LIN {X -62.6187,Y -12.3844,Z 71,A -174.9598,B 24.8879,C -2.444,E1 24.8427,E2 259.0842} C_DIS
LIN {X -63.2221,Y -8.7962,Z 71,A -178.5577,B 24.8875,C -2.4478,E1 24.8411,E2 262.6943} C_DIS
LIN {X -63.5633,Y -5.8378,Z 71,A 178.7584,B 24.8868,C -2.4559,E1 24.8403,E2 265.3749} C_DIS
LIN {X -63.7591,Y -3.0383,Z 71,A 176.0098,B 24.8865,C -2.4595,E1 24.8399,E2 268.1315} C_DIS
LIN {X -63.8232,Y 1.0014,Z 71,A 172.574,B 24.8851,C -2.4746,E1 24.8399,E2 271.552} C_DIS
LIN {X -63.7041,Y 4.0292,Z 71,A 169.9019,B 24.8842,C -2.484,E1 24.8402,E2 274.2176} C_DIS
LIN {X -63.478,Y 6.7017,Z 71,A 167.2312,B 24.8839,C -2.4868,E1 24.8409,E2 276.8978} C_DIS
LIN {X -62.7248,Y 11.8332,Z 71,A 163.1091,B 24.8816,C -2.5114,E1 24.8427,E2 280.9854} C_DIS
LIN {X -62.0016,Y 15.1714,Z 71,A 159.1214,B 24.8823,C -2.5038,E1 24.8452,E2 285.0149} C_DIS
LIN {X -61.1072,Y 18.4492,Z 71,A 156.1647,B 24.8813,C -2.5149,E1 24.8475,E2 287.9621} C_DIS
LIN {X -59.5419,Y 23.0056,Z 71,A 152.0273,B 24.8797,C -2.5315,E1 24.8514,E2 292.0832} C_DIS
LIN {X -57.4893,Y 27.7374,Z 71,A 147.1767,B 24.8788,C -2.5411,E1 24.857,E2 296.9374} C_DIS
LIN {X -55.3814,Y 31.7376,Z 71,A 143.5259,B 24.8769,C -2.5604,E1 24.8619,E2 300.5613} C_DIS
LIN {X -53.8615,Y 34.2546,Z 71,A 140.8267,B 24.8763,C -2.5666,E1 24.8658,E2 303.2594} C_DIS
LIN {X -51.327,Y 37.9471,Z 71,A 136.5857,B 24.8757,C -2.5733,E1 24.8727,E2 307.5055} C_DIS
LIN {X -49.8715,Y 39.8411,Z 71,A 134.6145,B 24.8748,C -2.5821,E1 24.8761,E2 309.4647} C_DIS
LIN {X -48.0177,Y 42.0557,Z 71,A 132.0307,B 24.8742,C -2.5889,E1 24.8807,E2 312.0442} C_DIS
LIN {X -46.1288,Y 44.1198,Z 71,A 129.2559,B 24.8741,C -2.5899,E1 24.8861,E2 314.8287} C_DIS
LIN {X -43.5524,Y 46.665,Z 71,A 126.2094,B 24.8729,C -2.6014,E1 24.8922,E2 317.8602} C_DIS
LIN {X -41.3478,Y 48.6285,Z 71,A 123.5743,B 24.8723,C -2.6076,E1 24.8977,E2 320.4909} C_DIS
LIN {X -39.1858,Y 50.3877,Z 71,A 120.9712,B 24.872,C -2.6109,E1 24.9034,E2 323.0959} C_DIS
LIN {X -36.3723,Y 52.4541,Z 71,A 117.5348,B 24.872,C -2.6112,E1 24.9112,E2 326.5435} C_DIS
LIN {X -33.3713,Y 54.4131,Z 71,A 114.6555,B 24.8707,C -2.6239,E1 24.918,E2 329.4017} C_DIS
LIN {X -30.7493,Y 55.9372,Z 71,A 111.9337,B 24.8703,C -2.6286,E1 24.9246,E2 332.1203} C_DIS
LIN {X -28.3087,Y 57.21,Z 71,A 109.4539,B 24.8699,C -2.6324,E1 24.9308,E2 334.5977} C_DIS
LIN {X -26.1605,Y 58.2237,Z 71,A 107.0088,B 24.8702,C -2.6292,E1 24.937,E2 337.0564} C_DIS
LIN {X -23.1449,Y 59.4872,Z 71,A 103.9447,B 24.8701,C -2.6305,E1 24.945,E2 340.1241} C_DIS
LIN {X -18.4974,Y 61.0929,Z 71,A 100.2418,B 24.8681,C -2.6504,E1 24.9547,E2 343.7865} C_DIS
LIN {X -15.1002,Y 62.019,Z 71,A 96.2614,B 24.8695,C -2.6364,E1 24.9655,E2 347.8059} C_DIS
LIN {X -10.983,Y 62.8796,Z 71,A 92.9646,B 24.8682,C -2.6494,E1 24.9745,E2 351.0755} C_DIS
LIN {X -7.8656,Y 63.3452,Z 71,A 89.7517,B 24.8688,C -2.643,E1 24.9834,E2 354.306} C_DIS
LIN {X -3.5629,Y 63.7313,Z 71,A 86.4625,B 24.8674,C -2.6573,E1 24.9925,E2 357.5625} C_DIS
LIN {X -1.027,Y 63.8227,Z 71,A 83.9639,B 24.8678,C -2.6532,E1 24.9995,E2 360.0713} C_DIS
LIN {X 1.838,Y 63.8044,Z 71,A 81.1896,B 24.8682,C -2.6491,E1 25.0073,E2 362.8548} C_DIS
LIN {X 5.3268,Y 63.6086,Z 71,A 78.2994,B 24.8677,C -2.6544,E1 25.0153,E2 365.7311} C_DIS
LIN {X 8.0773,Y 63.3178,Z 71,A 75.8118,B 24.8677,C -2.6539,E1 25.0222,E2 368.2182} C_DIS
LIN {X 10.8559,Y 62.9018,Z 71,A 72.9958,B 24.8685,C -2.6466,E1 25.03,E2 371.0488} C_DIS
LIN {X 14.3942,Y 62.1866,Z 71,A 69.0853,B 24.8701,C -2.6301,E1 25.0407,E2 374.993} C_DIS
LIN {X 17.9577,Y 61.253,Z 71,A 66.7167,B 24.8682,C -2.6489,E1 25.047,E2 377.3132} C_DIS
LIN {X 21.3417,Y 60.1569,Z 71,A 63.6072,B 24.8683,C -2.6482,E1 25.0552,E2 380.4184} C_DIS
LIN {X 24.1553,Y 59.0839,Z 71,A 60.6502,B 24.8692,C -2.6397,E1 25.0629,E2 383.3888} C_DIS
LIN {X 26.9211,Y 57.8759,Z 71,A 58.2592,B 24.8687,C -2.644,E1 25.0689,E2 385.7637} C_DIS
LIN {X 29.2585,Y 56.7306,Z 71,A 55.5229,B 24.8699,C -2.6318,E1 25.0758,E2 388.5214} C_DIS
LIN {X 32.7248,Y 54.8045,Z 71,A 52.3632,B 24.8695,C -2.6362,E1 25.0834,E2 391.6613} C_DIS
LIN {X 35.5421,Y 53.0209,Z 71,A 49.2654,B 24.8702,C -2.6291,E1 25.0907,E2 394.7658} C_DIS
LIN {X 38.8303,Y 50.6617,Z 71,A 46.138,B 24.8696,C -2.6349,E1 25.0977,E2 397.8683} C_DIS
LIN {X 40.4906,Y 49.3457,Z 71,A 43.4584,B 24.8718,C -2.6128,E1 25.1036,E2 400.5901} C_DIS
LIN {X 42.7839,Y 47.3708,Z 71,A 41.0277,B 24.8717,C -2.6144,E1 25.1087,E2 403.0075} C_DIS
LIN {X 44.9213,Y 45.3482,Z 71,A 38.4037,B 24.8722,C -2.6094,E1 25.1139,E2 405.6324} C_DIS
LIN {X 46.9119,Y 43.286,Z 71,A 35.417,B 24.8737,C -2.5938,E1 25.1197,E2 408.6428} C_DIS
LIN {X 49.423,Y 40.3956,Z 71,A 32.1479,B 24.8741,C -2.59,E1 25.1255,E2 411.906} C_DIS
LIN {X 51.6591,Y 37.4937,Z 71,A 29.1723,B 24.8741,C -2.5897,E1 25.1305,E2 414.868} C_DIS
LIN {X 53.729,Y 34.461,Z 71,A 26.1338,B 24.8743,C -2.5878,E1 25.1352,E2 417.8961} C_DIS
LIN {X 54.99,Y 32.4111,Z 71,A 23.8861,B 24.875,C -2.58,E1 25.1384,E2 420.1507} C_DIS
LIN {X 56.1908,Y 30.2818,Z 71,A 21.4597,B 24.8762,C -2.5684,E1 25.1417,E2 422.5918} C_DIS
LIN {X 57.4543,Y 27.8101,Z 71,A 18.594,B 24.8777,C -2.5523,E1 25.1453,E2 425.4802} C_DIS
LIN {X 58.9899,Y 24.3862,Z 71,A 15.8596,B 24.8771,C -2.5585,E1 25.1483,E2 428.1849} C_DIS
LIN {X 60.4513,Y 20.4944,Z 71,A 12.4555,B 24.8774,C -2.556,E1 25.1515,E2 431.5762} C_DIS
LIN {X 61.084,Y 18.5273,Z 71,A 10.1356,B 24.879,C -2.5388,E1 25.1535,E2 433.9235} C_DIS
LIN {X 62.2823,Y 13.9795,Z 71,A 5.8937,B 24.8803,C -2.5255,E1 25.1564,E2 438.1722} C_DIS
LIN {X 62.9014,Y 10.8581,Z 71,A 3.1608,B 24.8808,C -2.5199,E1 25.1578,E2 440.9025} C_DIS
LIN {X 63.3503,Y 7.8261,Z 71,A 0.3838,B 24.8817,C -2.5107,E1 25.1588,E2 443.6848} C_DIS
LIN {X 63.6624,Y 4.6453,Z 71,A -2.4692,B 24.8825,C -2.5021,E1 25.1595,E2 446.5412} C_DIS
LIN {X 63.7935,Y 2.1939,Z 71,A -4.6266,B 24.883,C -2.4963,E1 25.1597,E2 448.6994} C_DIS
LIN {X 63.8278,Y -0.7157,Z 71,A -7.2616,B 24.8839,C -2.4875,E1 25.1597,E2 451.3396} C_DIS
LIN {X 63.7474,Y -3.2705,Z 71,A -9.3744,B 24.8841,C -2.4848,E1 25.1595,E2 453.4461} C_DIS
LIN {X 63.5519,Y -5.9612,Z 71,A -11.9881,B 24.8853,C -2.4723,E1 25.1589,E2 456.0739} C_DIS
LIN {X 63.297,Y -8.2376,Z 71,A -13.9585,B 24.8857,C -2.4679,E1 25.1582,E2 458.043} C_DIS
LIN {X 62.8297,Y -11.2603,Z 71,A -16.6598,B 24.8864,C -2.4604,E1 25.157,E2 460.7463} C_DIS
LIN {X 62.2288,Y -14.2116,Z 71,A -19.8143,B 24.8882,C -2.4405,E1 25.155,E2 463.9294} C_DIS
LIN {X 61.2785,Y -17.8717,Z 71,A -23.5284,B 24.8899,C -2.422,E1 25.1522,E2 467.6661} C_DIS
LIN {X 60.2444,Y -21.0947,Z 71,A -25.546,B 24.8884,C -2.4383,E1 25.1504,E2 469.6335} C_DIS
LIN {X 59.3155,Y -23.5819,Z 71,A -28.0821,B 24.8894,C -2.4272,E1 25.1479,E2 472.1818} C_DIS
LIN {X 58.1993,Y -26.2147,Z 71,A -30.5908,B 24.89,C -2.421,E1 25.1451,E2 474.6915} C_DIS
LIN {X 56.3656,Y -29.9556,Z 71,A -34.4034,B 24.8912,C -2.4083,E1 25.1403,E2 478.5139} C_DIS
LIN {X 54.851,Y -32.6461,Z 71,A -37.0966,B 24.8917,C -2.4023,E1 25.1365,E2 481.2073} C_DIS
LIN {X 53.352,Y -35.042,Z 71,A -39.6135,B 24.8923,C -2.3958,E1 25.1327,E2 483.727} C_DIS
LIN {X 51.6176,Y -37.5502,Z 71,A -42.2132,B 24.8926,C -2.3918,E1 25.1285,E2 486.3235} C_DIS
LIN {X 50.3871,Y -39.1866,Z 71,A -44.5533,B 24.8942,C -2.3744,E1 25.1245,E2 488.6935} C_DIS
LIN {X 47.6744,Y -42.4447,Z 71,A -48.2527,B 24.8948,C -2.3674,E1 25.1177,E2 492.3928} C_DIS
LIN {X 44.4602,Y -45.8008,Z 71,A -51.9052,B 24.8946,C -2.3701,E1 25.1106,E2 496.0232} C_DIS
LIN {X 42.2771,Y -47.8242,Z 71,A -55.1278,B 24.8963,C -2.3505,E1 25.1039,E2 499.2794} C_DIS
LIN {X 38.6387,Y -50.809,Z 71,A -59.2519,B 24.8969,C -2.3439,E1 25.0949,E2 503.4038} C_DIS
LIN {X 36.16,Y -52.6015,Z 71,A -61.6657,B 24.8967,C -2.3464,E1 25.0894,E2 505.8032} C_DIS
LIN {X 33.2077,Y -54.5126,Z 71,A -65.1003,B 24.8978,C -2.3338,E1 25.0812,E2 509.2567} C_DIS
LIN {X 29.4719,Y -56.6204,Z 71,A -68.6212,B 24.8977,C -2.3351,E1 25.0726,E2 512.7644} C_DIS
LIN {X 27.1067,Y -57.7895,Z 71,A -71.1119,B 24.8983,C -2.3284,E1 25.0663,E2 515.2642} C_DIS
LIN {X 22.7062,Y -59.6558,Z 71,A -75.1549,B 24.8983,C -2.3282,E1 25.0559,E2 519.2985} C_DIS
LIN {X 20.3251,Y -60.5084,Z 71,A -77.5933,B 24.8989,C -2.3214,E1 25.0495,E2 521.7481} C_DIS
LIN {X 17.1942,Y -61.4717,Z 71,A -81.0111,B 24.9001,C -2.3071,E1 25.0402,E2 525.1941} C_DIS
LIN {X 13.4448,Y -62.399,Z 71,A -84.5829,B 24.9006,C -2.3015,E1 25.0305,E2 528.7743} C_DIS
LIN {X 9.3078,Y -63.1494,Z 71,A -87.811,B 24.8998,C -2.3112,E1 25.0216,E2 531.9762} C_DIS
LIN {X 6.2514,Y -63.5251,Z 71,A -90.5547,B 24.8998,C -2.31,E1 25.014,E2 534.7207} C_DIS
LIN {X 2.2633,Y -63.7909,Z 71,A -94.1016,B 24.8999,C -2.3095,E1 25.0041,E2 538.2675} C_DIS
LIN {X 2.2633,Y -63.7909,Z 71,A -94.1016,B 24.8999,C -2.3095,E1 25.0041,E2 538.2675} C_DIS
Enddeposition()
LIN {X 0.4088,Y -62.9103,Z 71,A -95.2964,B 24.8976,C -2.3357,E1 25.001,E2 539.4} C_DIS
Startdeposition()
$VEL.CP = VEL_PRINT
LIN {X 4.8964,Y -62.7212,Z 71,A -90.3905,B 24.8959,C -2.3556,E1 25.0148,E2 534.4483} C_DIS
LIN {X 7.9386,Y -62.4092,Z 71,A -87.6663,B 24.8959,C -2.3559,E1 25.0223,E2 531.7255} C_DIS
LIN {X 9.9278,Y -62.1244,Z 71,A -85.5507,B 24.8952,C -2.3638,E1 25.0282,E2 529.5932} C_DIS
LIN {X 14.3802,Y -61.2468,Z 71,A -81.6092,B 24.8952,C -2.363,E1 25.039,E2 525.6587} C_DIS
LIN {X 18.2735,Y -60.2001,Z 71,A -77.6153,B 24.8942,C -2.3746,E1 25.0497,E2 521.644} C_DIS
LIN {X 21.0359,Y -59.2912,Z 71,A -74.9878,B 24.8939,C -2.3774,E1 25.0567,E2 519.015} C_DIS
LIN {X 25.3175,Y -57.5931,Z 71,A -71.4757,B 24.8949,C -2.3671,E1 25.0656,E2 515.5357} C_DIS
LIN {X 27.5982,Y -56.5365,Z 71,A -68.883,B 24.8939,C -2.3779,E1 25.0722,E2 512.924} C_DIS
LIN {X 32.2402,Y -54.0234,Z 71,A -64.4511,B 24.8939,C -2.3771,E1 25.083,E2 508.5068} C_DIS
LIN {X 33.7475,Y -53.0951,Z 71,A -62.2788,B 24.8925,C -2.3938,E1 25.0882,E2 506.3021} C_DIS
LIN {X 36.1739,Y -51.4728,Z 71,A -60.1922,B 24.8933,C -2.3851,E1 25.093,E2 504.2432} C_DIS
LIN {X 38.2142,Y -49.9763,Z 71,A -57.4443,B 24.8918,C -2.4007,E1 25.0992,E2 501.4681} C_DIS
LIN {X 40.5717,Y -48.0823,Z 71,A -54.2934,B 24.8904,C -2.4166,E1 25.106,E2 498.2917} C_DIS
LIN {X 43.4852,Y -45.4643,Z 71,A -51.4365,B 24.8913,C -2.4072,E1 25.1117,E2 495.4687} C_DIS
LIN {X 45.7771,Y -43.1552,Z 71,A -48.2115,B 24.89,C -2.4209,E1 25.118,E2 492.2251} C_DIS
LIN {X 48.1586,Y -40.4806,Z 71,A -44.9232,B 24.8892,C -2.4299,E1 25.1241,E2 488.9305} C_DIS
LIN {X 50.3017,Y -37.7841,Z 71,A -41.8283,B 24.8885,C -2.4371,E1 25.1293,E2 485.8332} C_DIS
LIN {X 51.8685,Y -35.6047,Z 71,A -39.449,B 24.8881,C -2.4421,E1 25.1331,E2 483.4537} C_DIS
LIN {X 53.5761,Y -32.9793,Z 71,A -36.6728,B 24.8875,C -2.4482,E1 25.1373,E2 480.6773} C_DIS
LIN {X 54.635,Y -31.1922,Z 71,A -34.4713,B 24.8863,C -2.4614,E1 25.1403,E2 478.4558} C_DIS
LIN {X 56.2411,Y -28.1944,Z 71,A -31.9611,B 24.8868,C -2.4556,E1 25.1435,E2 475.9728} C_DIS
LIN {X 57.9933,Y -24.3862,Z 71,A -27.963,B 24.8854,C -2.4715,E1 25.1481,E2 471.9588} C_DIS
LIN {X 59.6027,Y -20.1352,Z 71,A -23.3656,B 24.8831,C -2.4958,E1 25.1525,E2 467.3297} C_DIS
LIN {X 60.5866,Y -16.9474,Z 71,A -19.8884,B 24.8811,C -2.5165,E1 25.1551,E2 463.8235} C_DIS
LIN {X 61.4837,Y -13.329,Z 71,A -17.5187,B 24.8826,C -2.5008,E1 25.1566,E2 461.5047} C_DIS
LIN {X 62.0144,Y -10.5908,Z 71,A -14.9926,B 24.8819,C -2.5084,E1 25.1578,E2 458.9754} C_DIS
LIN {X 62.2953,Y -8.7864,Z 71,A -12.8102,B 24.8801,C -2.527,E1 25.1587,E2 456.762} C_DIS
LIN {X 62.7823,Y -4.0411,Z 71,A -9.2522,B 24.8807,C -2.5206,E1 25.1595,E2 453.2401} C_DIS
LIN {X 62.8944,Y -1.5318,Z 71,A -6.7922,B 24.8796,C -2.5322,E1 25.1598,E2 450.7673} C_DIS
LIN {X 62.8961,Y 1.4392,Z 71,A -4.3486,B 24.8795,C -2.5341,E1 25.1598,E2 448.3337} C_DIS
LIN {X 62.7477,Y 4.5524,Z 71,A -1.161,B 24.8777,C -2.5519,E1 25.1592,E2 445.123} C_DIS
LIN {X 62.4375,Y 7.7199,Z 71,A 1.6878,B 24.877,C -2.5597,E1 25.1583,E2 442.2728} C_DIS
LIN {X 61.9807,Y 10.7901,Z 71,A 4.1459,B 24.877,C -2.5591,E1 25.1573,E2 439.8305} C_DIS
LIN {X 61.3864,Y 13.7751,Z 71,A 7.5,B 24.8748,C -2.5823,E1 25.1553,E2 436.4412} C_DIS
LIN {X 60.1896,Y 18.3094,Z 71,A 11.4443,B 24.8744,C -2.5867,E1 25.1523,E2 432.5089} C_DIS
LIN {X 58.8961,Y 22.1169,Z 71,A 14.7984,B 24.8741,C -2.5897,E1 25.1493,E2 429.1667} C_DIS
LIN {X 58.3235,Y 23.5859,Z 71,A 16.658,B 24.8727,C -2.6044,E1 25.1473,E2 427.2826} C_DIS
LIN {X 56.725,Y 27.2062,Z 71,A 20.3245,B 24.8715,C -2.616,E1 25.143,E2 423.6085} C_DIS
LIN {X 55.3285,Y 29.9445,Z 71,A 22.8764,B 24.8714,C -2.6173,E1 25.1397,E2 421.0669} C_DIS
LIN {X 53.8602,Y 32.5119,Z 71,A 25.5733,B 24.8707,C -2.6245,E1 25.1359,E2 418.3669} C_DIS
LIN {X 51.2918,Y 36.429,Z 71,A 29.6212,B 24.8701,C -2.6298,E1 25.1296,E2 414.3265} C_DIS
LIN {X 48.9356,Y 39.5376,Z 71,A 32.8944,B 24.87,C -2.6314,E1 25.1241,E2 411.065} C_DIS
LIN {X 47.6326,Y 41.0993,Z 71,A 35.4747,B 24.8678,C -2.6534,E1 25.1193,E2 408.4444} C_DIS
LIN {X 44.9625,Y 44.0042,Z 71,A 38.7622,B 24.8678,C -2.6537,E1 25.113,E2 405.1706} C_DIS
LIN {X 42.8337,Y 46.0794,Z 71,A 41.1397,B 24.868,C -2.6512,E1 25.1082,E2 402.8087} C_DIS
LIN {X 40.0841,Y 48.4891,Z 71,A 44.8355,B 24.8665,C -2.6663,E1 25.1004,E2 399.0916} C_DIS
LIN {X 38.1805,Y 50.0023,Z 71,A 47.9129,B 24.864,C -2.691,E1 25.0934,E2 395.967} C_DIS
LIN {X 35.2458,Y 52.1118,Z 71,A 50.7208,B 24.8646,C -2.6847,E1 25.087,E2 393.1835} C_DIS
LIN {X 32.0583,Y 54.1311,Z 71,A 53.6916,B 24.8653,C -2.6787,E1 25.08,E2 390.2361} C_DIS
LIN {X 29.279,Y 55.6835,Z 71,A 56.3613,B 24.8654,C -2.6772,E1 25.0735,E2 387.5777} C_DIS
LIN {X 26.6019,Y 57.0109,Z 71,A 59.2935,B 24.8646,C -2.6854,E1 25.0661,E2 384.6338} C_DIS
LIN {X 23.5561,Y 58.3346,Z 71,A 62.2303,B 24.8645,C -2.6865,E1 25.0585,E2 381.7012} C_DIS
LIN {X 20.5285,Y 59.4683,Z 71,A 65.5611,B 24.8633,C -2.698,E1 25.0497,E2 378.35} C_DIS
LIN {X 17.7095,Y 60.3682,Z 71,A 67.8415,B 24.8641,C -2.6905,E1 25.0437,E2 376.0915} C_DIS
LIN {X 13.446,Y 61.4582,Z 71,A 71.6552,B 24.8643,C -2.6884,E1 25.0334,E2 372.2885} C_DIS
LIN {X 10.0786,Y 62.1001,Z 71,A 75.0149,B 24.8636,C -2.6948,E1 25.0241,E2 368.9172} C_DIS
LIN {X 7.2724,Y 62.4902,Z 71,A 77.6363,B 24.8635,C -2.6963,E1 25.0168,E2 366.2944} C_DIS
LIN {X 3.3459,Y 62.823,Z 71,A 81.6983,B 24.8624,C -2.7068,E1 25.0055,E2 362.2092} C_DIS
LIN {X -0.8066,Y 62.9077,Z 71,A 85.0123,B 24.8635,C -2.6958,E1 24.9963,E2 358.9215} C_DIS
LIN {X -3.3309,Y 62.8238,Z 71,A 87.9825,B 24.8621,C -2.7096,E1 24.9879,E2 355.9178} C_DIS
LIN {X -7.6361,Y 62.4476,Z 71,A 91.4384,B 24.8634,C -2.6971,E1 24.9784,E2 352.4895} C_DIS
LIN {X -11.4181,Y 61.8677,Z 71,A 94.4374,B 24.8647,C -2.6843,E1 24.9702,E2 349.5181} C_DIS
LIN {X -14.7659,Y 61.1547,Z 71,A 98.3814,B 24.8632,C -2.699,E1 24.9594,E2 345.534} C_DIS
LIN {X -18.0979,Y 60.2529,Z 71,A 101.4372,B 24.8637,C -2.6938,E1 24.9512,E2 342.4857} C_DIS
LIN {X -22.5115,Y 58.7469,Z 71,A 105.075,B 24.8655,C -2.6758,E1 24.9417,E2 338.8835} C_DIS
LIN {X -24.4313,Y 57.9743,Z 71,A 107.2309,B 24.8652,C -2.6788,E1 24.9361,E2 336.7156} C_DIS
LIN {X -27.469,Y 56.5988,Z 71,A 109.9857,B 24.8663,C -2.6684,E1 24.9292,E2 333.9786} C_DIS
LIN {X -29.8101,Y 55.4014,Z 71,A 112.6392,B 24.8662,C -2.6698,E1 24.9226,E2 331.3146} C_DIS
LIN {X -32.3659,Y 53.9489,Z 71,A 115.1019,B 24.8671,C -2.6607,E1 24.9167,E2 328.8661} C_DIS
LIN {X -35.9826,Y 51.6058,Z 71,A 119.7528,B 24.8664,C -2.6678,E1 24.9058,E2 324.1829} C_DIS
LIN {X -39.3053,Y 49.1237,Z 71,A 123.0518,B 24.8681,C -2.6503,E1 24.8986,E2 320.9135} C_DIS
LIN {X -41.5853,Y 47.2085,Z 71,A 125.6154,B 24.869,C -2.6415,E1 24.8932,E2 318.3612} C_DIS
LIN {X -44.217,Y 44.7522,Z 71,A 129.6208,B 24.8683,C -2.6481,E1 24.8851,E2 314.3231} C_DIS
LIN {X -47.1286,Y 41.6765,Z 71,A 132.9522,B 24.8703,C -2.6283,E1 24.8789,E2 311.0244} C_DIS
LIN {X -49.169,Y 39.2481,Z 71,A 136.4415,B 24.8699,C -2.6326,E1 24.8727,E2 307.5087} C_DIS
LIN {X -51.4058,Y 36.2693,Z 71,A 139.0685,B 24.8722,C -2.6087,E1 24.8684,E2 304.926} C_DIS
LIN {X -53.397,Y 33.2667,Z 71,A 142.5812,B 24.8727,C -2.6041,E1 24.8631,E2 301.4065} C_DIS
LIN {X -54.8842,Y 30.7513,Z 71,A 145.0912,B 24.8737,C -2.5937,E1 24.8596,E2 298.9084} C_DIS
LIN {X -56.6546,Y 27.3528,Z 71,A 149.2957,B 24.8734,C -2.5972,E1 24.8543,E2 294.6729} C_DIS
LIN {X -58.8083,Y 22.3493,Z 71,A 154.0448,B 24.8752,C -2.5782,E1 24.8493,E2 289.9427} C_DIS
LIN {X -60.0926,Y 18.6223,Z 71,A 157.4276,B 24.8767,C -2.5633,E1 24.8464,E2 286.5762} C_DIS
LIN {X -61.0033,Y 15.3812,Z 71,A 160.6071,B 24.8774,C -2.5559,E1 24.8441,E2 283.3958} C_DIS
LIN {X -61.7487,Y 12.0428,Z 71,A 163.3403,B 24.879,C -2.539,E1 24.8425,E2 280.6871} C_DIS
LIN {X -62.3275,Y 8.5559,Z 71,A 166.484,B 24.8801,C -2.5274,E1 24.8412,E2 277.5523} C_DIS
LIN {X -62.7001,Y 5.1605,Z 71,A 169.9296,B 24.8804,C -2.5238,E1 24.8402,E2 274.0946} C_DIS
LIN {X -62.8727,Y 2.2431,Z 71,A 172.9217,B 24.8806,C -2.5216,E1 24.8398,E2 271.0897} C_DIS
LIN {X -62.8997,Y -1.2436,Z 71,A 175.7407,B 24.8822,C -2.5049,E1 24.8398,E2 268.2937} C_DIS
LIN {X -62.7846,Y -4.0074,Z 71,A 178.3432,B 24.8828,C -2.4986,E1 24.8402,E2 265.6908} C_DIS
LIN {X -62.5283,Y -6.9462,Z 71,A -179.0365,B 24.8837,C -2.4889,E1 24.8409,E2 263.0778} C_DIS
LIN {X -61.7486,Y -12.0434,Z 71,A -174.3261,B 24.8851,C -2.4747,E1 24.8431,E2 258.3733} C_DIS
LIN {X -61.135,Y -14.8466,Z 71,A -171.4136,B 24.8853,C -2.4725,E1 24.8449,E2 255.4491} C_DIS
LIN {X -60.3399,Y -17.8048,Z 71,A -169.0172,B 24.8867,C -2.4566,E1 24.8467,E2 253.0766} C_DIS
LIN {X -59.0357,Y -21.7425,Z 71,A -164.8952,B 24.8871,C -2.4522,E1 24.8504,E2 248.9418} C_DIS
LIN {X -57.967,Y -24.4486,Z 71,A -162.2124,B 24.8878,C -2.4453,E1 24.8532,E2 246.2605} C_DIS
LIN {X -56.1817,Y -28.3134,Z 71,A -158.3146,B 24.8887,C -2.435,E1 24.8579,E2 242.3662} C_DIS
LIN {X -54.7385,Y -31.012,Z 71,A -155.8542,B 24.89,C -2.4212,E1 24.8612,E2 239.9257} C_DIS
LIN {X -53.3545,Y -33.3348,Z 71,A -153.1524,B 24.8901,C -2.4195,E1 24.8651,E2 237.214} C_DIS
LIN {X -52.1891,Y -35.1317,Z 71,A -151.04,B 24.8903,C -2.4178,E1 24.8684,E2 235.0952} C_DIS
LIN {X -50.5083,Y -37.5092,Z 71,A -148.1197,B 24.8903,C -2.4167,E1 24.8732,E2 232.1634} C_DIS
LIN {X -47.7584,Y -40.9522,Z 71,A -143.9738,B 24.891,C -2.4102,E1 24.8806,E2 228.0139} C_DIS
LIN {X -45.4246,Y -43.5264,Z 71,A -140.4594,B 24.891,C -2.4105,E1 24.8874,E2 224.4835} C_DIS
LIN {X -43.1321,Y -45.7988,Z 71,A -138.2164,B 24.8928,C -2.3904,E1 24.8919,E2 222.2792} C_DIS
LIN {X -40.992,Y -47.7245,Z 71,A -135.9085,B 24.8938,C -2.379,E1 24.8967,E2 219.9894} C_DIS
LIN {X -38.0442,Y -50.1063,Z 71,A -132.1643,B 24.8938,C -2.3788,E1 24.9049,E2 216.2318} C_DIS
LIN {X -35.4238,Y -51.9913,Z 71,A -129.208,B 24.8942,C -2.3743,E1 24.9117,E2 213.276} C_DIS
LIN {X -32.9401,Y -53.5999,Z 71,A -126.4883,B 24.8945,C -2.3708,E1 24.9181,E2 210.556} C_DIS
LIN {X -29.5358,Y -55.5482,Z 71,A -122.8143,B 24.8948,C -2.3681,E1 24.9271,E2 206.8777} C_DIS
LIN {X -26.3368,Y -57.1332,Z 71,A -119.7532,B 24.8955,C -2.3604,E1 24.9347,E2 203.8273} C_DIS
LIN {X -23.4448,Y -58.3802,Z 71,A -116.5011,B 24.895,C -2.3657,E1 24.9432,E2 200.5552} C_DIS
LIN {X -20.6961,Y -59.4104,Z 71,A -114.3067,B 24.8961,C -2.3531,E1 24.9489,E2 198.3864} C_DIS
LIN {X -16.4933,Y -60.7115,Z 71,A -110.3889,B 24.8965,C -2.3484,E1 24.9594,E2 194.4731} C_DIS
LIN {X -13.2097,Y -61.5098,Z 71,A -107.0373,B 24.8961,C -2.3528,E1 24.9685,E2 191.1066} C_DIS
LIN {X -10.4504,Y -62.0379,Z 71,A -104.5189,B 24.8963,C -2.3511,E1 24.9754,E2 188.5897} C_DIS
LIN {X -8.4287,Y -62.3457,Z 71,A -102.3451,B 24.8957,C -2.3576,E1 24.9815,E2 186.3989} C_DIS
LIN {X -4.1146,Y -62.7773,Z 71,A -98.688,B 24.8963,C -2.3509,E1 24.9916,E2 182.7558} C_DIS
LIN {X -1.4104,Y -62.8966,Z 71,A -96.2627,B 24.8963,C -2.3503,E1 24.9984,E2 180.3316} C_DIS
LIN {X 0.4088,Y -62.9103,Z 71,A -95.2953,B 24.8977,C -2.3352,E1 25.001,E2 179.4} C_DIS
Enddeposition()
LIN {X 0.4088,Y -62.9103,Z 71,A -95.2953,B 24.8977,C -2.3352,E1 25.001,E2 179.4} C_DIS
Startdeposition()
$VEL.CP = VEL_PRINT
LIN {X 0.3113,Y -61.9923,Z 71,A -95.9555,B 24.8974,C -2.3387,E1 24.9992,E2 180.052} C_DIS
LIN {X -2.6969,Y -61.9343,Z 71,A -98.6873,B 24.8974,C -2.3394,E1 24.9915,E2 182.7826} C_DIS
LIN {X -4.8385,Y -61.8036,Z 71,A -101.7441,B 24.8993,C -2.3166,E1 24.9829,E2 185.8949} C_DIS
LIN {X -8.674,Y -61.3832,Z 71,A -103.9917,B 24.8968,C -2.3451,E1 24.9768,E2 188.0763} C_DIS
LIN {X -10.8761,Y -61.0316,Z 71,A -106.2994,B 24.8972,C -2.3405,E1 24.9704,E2 190.3972} C_DIS
LIN {X -15.6813,Y -59.9775,Z 71,A -111.1152,B 24.8975,C -2.3371,E1 24.9573,E2 195.2274} C_DIS
LIN {X -19.8959,Y -58.7137,Z 71,A -114.6912,B 24.8964,C -2.3502,E1 24.9478,E2 198.7785} C_DIS
LIN {X -21.6548,Y -58.0886,Z 71,A -116.849,B 24.897,C -2.3428,E1 24.9421,E2 200.9582} C_DIS
LIN {X -24.828,Y -56.8041,Z 71,A -119.7404,B 24.8962,C -2.3516,E1 24.9347,E2 203.8354} C_DIS
LIN {X -27.3149,Y -55.6515,Z 71,A -122.6661,B 24.8967,C -2.3466,E1 24.9273,E2 206.7805} C_DIS
LIN {X -31.8411,Y -53.1921,Z 71,A -127.1895,B 24.8957,C -2.3578,E1 24.9163,E2 211.2904} C_DIS
LIN {X -34.2462,Y -51.6755,Z 71,A -129.8643,B 24.8954,C -2.3609,E1 24.9101,E2 213.9665} C_DIS
LIN {X -36.9284,Y -49.795,Z 71,A -132.7409,B 24.8947,C -2.3689,E1 24.9036,E2 216.8341} C_DIS
LIN {X -39.8094,Y -47.5227,Z 71,A -136.3028,B 24.8945,C -2.3717,E1 24.8958,E2 220.4026} C_DIS
LIN {X -42.499,Y -45.1328,Z 71,A -139.8418,B 24.8942,C -2.3741,E1 24.8885,E2 223.9501} C_DIS
LIN {X -44.8507,Y -42.7977,Z 71,A -142.9761,B 24.8938,C -2.3792,E1 24.8824,E2 227.0858} C_DIS
LIN {X -47.251,Y -40.1308,Z 71,A -145.9762,B 24.8926,C -2.3926,E1 24.8769,E2 230.0673} C_DIS
LIN {X -49.7312,Y -37.0137,Z 71,A -149.401,B 24.8914,C -2.4061,E1 24.871,E2 233.4761} C_DIS
LIN {X -51.211,Y -34.9373,Z 71,A -152.0185,B 24.8913,C -2.407,E1 24.8668,E2 236.1043} C_DIS
LIN {X -53.1635,Y -31.8887,Z 71,A -155.4479,B 24.8906,C -2.414,E1 24.8617,E2 239.5345} C_DIS
LIN {X -54.1916,Y -30.1068,Z 71,A -157.3431,B 24.8902,C -2.4191,E1 24.8592,E2 241.4273} C_DIS
LIN {X -55.7759,Y -27.0599,Z 71,A -160.5973,B 24.8895,C -2.4263,E1 24.8551,E2 244.6819} C_DIS
LIN {X -57.2748,Y -23.7247,Z 71,A -163.6284,B 24.8881,C -2.4422,E1 24.8517,E2 247.6917} C_DIS
LIN {X -58.0912,Y -21.6484,Z 71,A -166.7153,B 24.8892,C -2.4294,E1 24.8486,E2 250.8266} C_DIS
LIN {X -59.4153,Y -17.6905,Z 71,A -170.1094,B 24.8874,C -2.4491,E1 24.8458,E2 254.193} C_DIS
LIN {X -60.3121,Y -14.3405,Z 71,A -173.2308,B 24.8864,C -2.4603,E1 24.8437,E2 257.306} C_DIS
LIN {X -60.824,Y -11.9851,Z 71,A -175.5845,B 24.886,C -2.4648,E1 24.8424,E2 259.6628} C_DIS
LIN {X -61.5813,Y -7.1329,Z 71,A -179.4554,B 24.8835,C -2.491,E1 24.8408,E2 263.4942} C_DIS
LIN {X -61.7758,Y -5.1916,Z 71,A 177.8547,B 24.8845,C -2.4806,E1 24.8401,E2 266.2252} C_DIS
LIN {X -61.9779,Y -1.3896,Z 71,A 174.5261,B 24.8832,C -2.4951,E1 24.8398,E2 269.5392} C_DIS
LIN {X -61.9272,Y 2.8618,Z 71,A 170.6768,B 24.8818,C -2.5089,E1 24.8401,E2 273.3785} C_DIS
LIN {X -61.6929,Y 6.0965,Z 71,A 167.7344,B 24.8809,C -2.5194,E1 24.8407,E2 276.3136} C_DIS
LIN {X -61.3572,Y 8.8572,Z 71,A 165.1204,B 24.8802,C -2.5267,E1 24.8417,E2 278.9256} C_DIS
LIN {X -60.858,Y 11.8088,Z 71,A 161.6038,B 24.8806,C -2.522,E1 24.8435,E2 282.4743} C_DIS
LIN {X -59.9913,Y 15.6276,Z 71,A 158.9891,B 24.8778,C -2.5513,E1 24.8452,E2 285.0344} C_DIS
LIN {X -59.4261,Y 17.6543,Z 71,A 156.8691,B 24.8775,C -2.5541,E1 24.8469,E2 287.1599} C_DIS
LIN {X -58.6281,Y 20.1476,Z 71,A 154.2259,B 24.8772,C -2.5575,E1 24.8492,E2 289.8101} C_DIS
LIN {X -56.6918,Y 25.0856,Z 71,A 149.5316,B 24.8754,C -2.5759,E1 24.8541,E2 294.4865} C_DIS
LIN {X -55.9421,Y 26.7139,Z 71,A 147.3047,B 24.876,C -2.5705,E1 24.8568,E2 296.7386} C_DIS
LIN {X -53.6699,Y 31.0275,Z 71,A 143.2889,B 24.8738,C -2.5923,E1 24.8621,E2 300.7234} C_DIS
LIN {X -52.0224,Y 33.7176,Z 71,A 139.9977,B 24.8738,C -2.5935,E1 24.867,E2 304.0284} C_DIS
LIN {X -50.385,Y 36.1179,Z 71,A 136.5154,B 24.8744,C -2.5862,E1 24.8728,E2 307.5452} C_DIS
LIN {X -48.1281,Y 39.0746,Z 71,A 134.0686,B 24.8718,C -2.6133,E1 24.8769,E2 309.9388} C_DIS
LIN {X -46.2595,Y 41.2699,Z 71,A 131.0583,B 24.8718,C -2.6135,E1 24.8825,E2 312.9621} C_DIS
LIN {X -43.6686,Y 44.0023,Z 71,A 127.8518,B 24.8704,C -2.627,E1 24.8887,E2 316.1502} C_DIS
LIN {X -41.2002,Y 46.3219,Z 71,A 125.0265,B 24.8691,C -2.6399,E1 24.8944,E2 318.9561} C_DIS
LIN {X -39.4055,Y 47.8583,Z 71,A 122.5548,B 24.8692,C -2.6392,E1 24.8998,E2 321.4391} C_DIS
LIN {X -36.7727,Y 49.9092,Z 71,A 119.4513,B 24.8686,C -2.6452,E1 24.9066,E2 324.5394} C_DIS
LIN {X -33.8428,Y 51.9401,Z 71,A 115.6943,B 24.8689,C -2.6427,E1 24.9154,E2 328.3149} C_DIS
LIN {X -30.5709,Y 53.9319,Z 71,A 112.2248,B 24.8681,C -2.6503,E1 24.9237,E2 331.7767} C_DIS
LIN {X -26.8509,Y 55.8763,Z 71,A 108.8416,B 24.8665,C -2.6661,E1 24.9321,E2 335.1311} C_DIS
LIN {X -24.6603,Y 56.8772,Z 71,A 106.4113,B 24.8665,C -2.6654,E1 24.9383,E2 337.5691} C_DIS
LIN {X -21.8766,Y 58.0048,Z 71,A 103.5177,B 24.8665,C -2.6667,E1 24.9459,E2 340.4657} C_DIS
LIN {X -18.3017,Y 59.2299,Z 71,A 100.439,B 24.8652,C -2.6791,E1 24.954,E2 343.5206} C_DIS
LIN {X -16.6693,Y 59.7103,Z 71,A 98.4965,B 24.8658,C -2.6733,E1 24.9592,E2 345.48} C_DIS
LIN {X -13.3355,Y 60.5418,Z 71,A 95.4894,B 24.8652,C -2.6796,E1 24.9674,E2 348.4761} C_DIS
LIN {X -10.7838,Y 61.048,Z 71,A 92.5359,B 24.8661,C -2.6703,E1 24.9755,E2 351.4548} C_DIS
LIN {X -7.1248,Y 61.5823,Z 71,A 88.4424,B 24.8673,C -2.6585,E1 24.987,E2 355.5791} C_DIS
LIN {X -3.0989,Y 61.9163,Z 71,A 86.1409,B 24.8642,C -2.6895,E1 24.9932,E2 357.8078} C_DIS
LIN {X -0.9425,Y 61.9862,Z 71,A 83.4829,B 24.8655,C -2.6761,E1 25.0007,E2 360.4978} C_DIS
LIN {X 2.8478,Y 61.9278,Z 71,A 79.6178,B 24.8662,C -2.6689,E1 25.0115,E2 364.3791} C_DIS
LIN {X 7.4433,Y 61.545,Z 71,A 76.075,B 24.8648,C -2.6836,E1 25.0213,E2 367.8848} C_DIS
LIN {X 11.1818,Y 60.9766,Z 71,A 72.6331,B 24.8648,C -2.6836,E1 25.0307,E2 371.323} C_DIS
LIN {X 14.0147,Y 60.3881,Z 71,A 69.2149,B 24.8665,C -2.6662,E1 25.0401,E2 374.7779} C_DIS
LIN {X 17.8059,Y 59.3811,Z 71,A 66.5405,B 24.8647,C -2.6845,E1 25.0472,E2 377.4045} C_DIS
LIN {X 20.4254,Y 58.5316,Z 71,A 63.6496,B 24.8656,C -2.6748,E1 25.0549,E2 380.3129} C_DIS
LIN {X 23.1515,Y 57.5076,Z 71,A 61.0572,B 24.8656,C -2.6744,E1 25.0616,E2 382.9005} C_DIS
LIN {X 26.2828,Y 56.1459,Z 71,A 57.4513,B 24.8671,C -2.6608,E1 25.0709,E2 386.5296} C_DIS
LIN {X 29.1186,Y 54.7294,Z 71,A 54.9718,B 24.8664,C -2.6671,E1 25.077,E2 388.9872} C_DIS
LIN {X 31.868,Y 53.1761,Z 71,A 51.6687,B 24.8677,C -2.6543,E1 25.085,E2 392.3106} C_DIS
LIN {X 35.0504,Y 51.1344,Z 71,A 47.8961,B 24.8689,C -2.6424,E1 25.0937,E2 396.0988} C_DIS
LIN {X 38.0675,Y 48.9294,Z 71,A 44.8723,B 24.8685,C -2.6462,E1 25.1004,E2 399.1027} C_DIS
LIN {X 41.2487,Y 46.2784,Z 71,A 40.829,B 24.8697,C -2.6339,E1 25.109,E2 403.1592} C_DIS
LIN {X 45.6061,Y 41.9908,Z 71,A 35.649,B 24.8698,C -2.6329,E1 25.1191,E2 408.3193} C_DIS
LIN {X 47.9463,Y 39.2988,Z 71,A 32.7773,B 24.8696,C -2.6355,E1 25.1242,E2 411.1719} C_DIS
LIN {X 50.2275,Y 36.3381,Z 71,A 29.318,B 24.8704,C -2.6271,E1 25.1301,E2 414.6346} C_DIS
LIN {X 52.4114,Y 33.11,Z 71,A 25.5055,B 24.8718,C -2.613,E1 25.136,E2 418.4615} C_DIS
LIN {X 53.7336,Y 30.9166,Z 71,A 22.9143,B 24.8729,C -2.6014,E1 25.1397,E2 421.0668} C_DIS
LIN {X 56.0469,Y 26.4956,Z 71,A 18.1407,B 24.8746,C -2.5849,E1 25.1457,E2 425.8539} C_DIS
LIN {X 57.4497,Y 23.2954,Z 71,A 15.0182,B 24.8752,C -2.5784,E1 25.1491,E2 428.9748} C_DIS
LIN {X 58.9758,Y 19.1046,Z 71,A 11.5922,B 24.8747,C -2.5834,E1 25.1522,E2 432.3698} C_DIS
LIN {X 59.8852,Y 16.0286,Z 71,A 7.7831,B 24.8776,C -2.5539,E1 25.1552,E2 436.2267} C_DIS
LIN {X 61.0888,Y 10.555,Z 71,A 3.0456,B 24.878,C -2.5489,E1 25.1578,E2 440.9485} C_DIS
LIN {X 61.5247,Y 7.6136,Z 71,A 0.3516,B 24.8787,C -2.5417,E1 25.1588,E2 443.6436} C_DIS
LIN {X 61.833,Y 4.4595,Z 71,A -3.2053,B 24.8811,C -2.5171,E1 25.1596,E2 447.2374} C_DIS
LIN {X 61.9903,Y 0.6775,Z 71,A -5.9984,B 24.8805,C -2.5234,E1 25.1598,E2 449.9991} C_DIS
LIN {X 61.9529,Y -2.2583,Z 71,A -8.7076,B 24.8813,C -2.5149,E1 25.1596,E2 452.7122} C_DIS
LIN {X 61.7793,Y -5.1426,Z 71,A -11.2282,B 24.8817,C -2.5101,E1 25.1591,E2 455.2291} C_DIS
LIN {X 61.4764,Y -7.9865,Z 71,A -14.1731,B 24.8832,C -2.4943,E1 25.1581,E2 458.194} C_DIS
LIN {X 61.0452,Y -10.8,Z 71,A -16.6076,B 24.8835,C -2.4909,E1 25.157,E2 460.6223} C_DIS
LIN {X 60.2075,Y -14.7716,Z 71,A -20.7687,B 24.8856,C -2.4691,E1 25.1544,E2 464.8109} C_DIS
LIN {X 58.8817,Y -19.3913,Z 71,A -24.7637,B 24.8858,C -2.4663,E1 25.1512,E2 468.7895} C_DIS
LIN {X 58.0197,Y -21.8371,Z 71,A -26.9787,B 24.8861,C -2.4635,E1 25.1491,E2 470.9989} C_DIS
LIN {X 57.0591,Y -24.2367,Z 71,A -30.2528,B 24.8887,C -2.4347,E1 25.1455,E2 474.3229} C_DIS
LIN {X 55.7291,Y -27.1572,Z 71,A -32.3779,B 24.8877,C -2.4464,E1 25.143,E2 476.4089} C_DIS
LIN {X 53.6661,Y -31.0341,Z 71,A -36.474,B 24.8888,C -2.4338,E1 25.1375,E2 480.5134} C_DIS
LIN {X 52.1753,Y -33.4794,Z 71,A -39.2137,B 24.8897,C -2.4242,E1 25.1334,E2 483.2621} C_DIS
LIN {X 49.6634,Y -37.104,Z 71,A -42.9964,B 24.8901,C -2.4203,E1 25.1273,E2 487.0356} C_DIS
LIN {X 48.3641,Y -38.7834,Z 71,A -45.1686,B 24.891,C -2.41,E1 25.1235,E2 489.2218} C_DIS
LIN {X 46.399,Y -41.114,Z 71,A -48.0006,B 24.8917,C -2.4025,E1 25.1184,E2 492.0587} C_DIS
LIN {X 44.1032,Y -43.5665,Z 71,A -50.7349,B 24.8916,C -2.4039,E1 25.1131,E2 494.778} C_DIS
LIN {X 42.8424,Y -44.8076,Z 71,A -52.78,B 24.8928,C -2.3902,E1 25.109,E2 496.847} C_DIS
LIN {X 40.3893,Y -47.0308,Z 71,A -55.8479,B 24.8934,C -2.3831,E1 25.1025,E2 499.9196} C_DIS
LIN {X 37.8065,Y -49.1305,Z 71,A -58.7411,B 24.8936,C -2.3808,E1 25.0962,E2 502.8072} C_DIS
LIN {X 35.7444,Y -50.6515,Z 71,A -60.9851,B 24.8938,C -2.3789,E1 25.0911,E2 505.0479} C_DIS
LIN {X 32.7537,Y -52.634,Z 71,A -63.9145,B 24.8936,C -2.3817,E1 25.0843,E2 507.9611} C_DIS
LIN {X 29.0053,Y -54.789,Z 71,A -67.8559,B 24.8941,C -2.3759,E1 25.0748,E2 511.9045} C_DIS
LIN {X 24.9909,Y -56.7331,Z 71,A -72.382,B 24.8955,C -2.36,E1 25.0633,E2 516.4563} C_DIS
LIN {X 22.6731,Y -57.698,Z 71,A -74.8671,B 24.8961,C -2.353,E1 25.0568,E2 518.9524} C_DIS
LIN {X 20.2386,Y -58.5967,Z 71,A -77.7474,B 24.8973,C -2.3391,E1 25.0492,E2 521.86} C_DIS
LIN {X 14.9591,Y -60.1617,Z 71,A -82.9113,B 24.898,C -2.3321,E1 25.0352,E2 527.0322} C_DIS
LIN {X 9.2228,Y -61.3036,Z 71,A -87.4872,B 24.8967,C -2.3463,E1 25.0228,E2 531.5694} C_DIS
LIN {X 4.6894,Y -61.8159,Z 71,A -91.8319,B 24.8972,C -2.3411,E1 25.0107,E2 535.9235} C_DIS
LIN {X 0.3813,Y -61.9902,Z 71,A -93.9308,B 24.8936,C -2.3816,E1 25.0051,E2 537.9255} C_DIS
Enddeposition()
LIN {X 0.3813,Y -61.9902,Z 71,A -93.9308,B 24.8936,C -2.3816,E1 25.0051,E2 537.9255} C_DIS
Startdeposition()
$VEL.CP = VEL_PRINT
LIN {X 3.9598,Y -60.9458,Z 71,A -91.7532,B 24.8944,C -2.3722,E1 25.0111,E2 535.7709} C_DIS
LIN {X 7.0018,Y -60.6713,Z 71,A -88.1136,B 24.8927,C -2.3909,E1 25.0213,E2 532.0892} C_DIS
Enddeposition()
END
